LIN {X 0,Y 488.816,Z 673.843,A -85,B 0,C 180,E1 23597.214,E2 23597.214} C_VEL
LIN {X 0,Y 488.827,Z 673.82,A -85,B 0,C 180,E1 23593.605,E2 23593.605} C_VEL
LIN {X 0,Y 488.821,Z 673.843,A -85,B 0,C 180,E1 23590.012,E2 23590.012} C_VEL
LIN {X 0,Y 488.815,Z 673.84,A -85,B 0,C 180,E1 23586.459,E2 23586.459} C_VEL
LIN {X 0,Y 488.829,Z 673.833,A -85,B 0,C 180,E1 23582.931,E2 23582.931} C_VEL
LIN {X 0,Y 488.826,Z 673.843,A -85,B 0,C 180,E1 23579.297,E2 23579.297} C_VEL
LIN {X 0,Y 488.815,Z 673.842,A -85,B 0,C 180,E1 23575.659,E2 23575.659} C_VEL
LIN {X 0,Y 488.835,Z 673.84,A -85,B 0,C 180,E1 23572.123,E2 23572.123} C_VEL
LIN {X 0,Y 488.826,Z 673.833,A -85,B 0,C 180,E1 23568.556,E2 23568.556} C_VEL
LIN {X 0,Y 488.817,Z 673.838,A -85,B 0,C 180,E1 23564.943,E2 23564.943} C_VEL
LIN {X 0,Y 488.831,Z 673.84,A -85,B 0,C 180,E1 23561.392,E2 23561.392} C_VEL
LIN {X 0,Y 488.831,Z 673.844,A -85,B 0,C 180,E1 23557.765,E2 23557.765} C_VEL
LIN {X 0,Y 488.817,Z 673.841,A -85,B 0,C 180,E1 23554.155,E2 23554.155} C_VEL
LIN {X 0,Y 488.824,Z 673.804,A -85,B 0,C 180,E1 23550.6,E2 23550.6} C_VEL
LIN {X 0,Y 488.83,Z 673.841,A -85,B 0,C 180,E1 23546.992,E2 23546.992} C_VEL
LIN {X 0,Y 488.813,Z 673.808,A -85,B 0,C 180,E1 23543.47,E2 23543.47} C_VEL
LIN {X 0,Y 488.822,Z 673.844,A -85,B 0,C 180,E1 23539.885,E2 23539.885} C_VEL
LIN {X 0,Y 488.822,Z 673.817,A -85,B 0,C 180,E1 23536.221,E2 23536.221} C_VEL
LIN {X 0,Y 488.818,Z 673.811,A -85,B 0,C 180,E1 23532.75,E2 23532.75} C_VEL
LIN {X 0,Y 488.863,Z 674.082,A -85,B 0,C 180,E1 23530.778,E2 23530.778} C_VEL
LIN {X 0,Y 489.222,Z 675.525,A -85,B 0,C 180,E1 23530.578,E2 23530.578} C_VEL
LIN {X 0,Y 491.282,Z 678.683,A -85,B 0,C 180,E1 23530.298,E2 23530.298} C_VEL
LIN {X 0,Y 492.455,Z 680.416,A -85,B 0,C 180,E1 23530.144,E2 23530.144} C_VEL
LIN {X 0,Y 504.755,Z 699.098,A -85,B 0,C 180,E1 23528.583,E2 23528.583} C_VEL
LIN {X 0,Y 508.963,Z 706.354,A -85,B 0,C 180,E1 23528.059,E2 23528.059} C_VEL
LIN {X 0,Y 508.656,Z 723.177,A -85,B 0,C 180,E1 23527.787,E2 23527.787} C_VEL
LIN {X 0,Y 507.74,Z 730.874,A -85,B 0,C 180,E1 23527.733,E2 23527.733} C_VEL
LIN {X 0,Y 502.491,Z 751.441,A -85,B 0,C 180,E1 23527.848,E2 23527.848} C_VEL
LIN {X 0,Y 501.776,Z 758.046,A -85,B 0,C 180,E1 23527.795,E2 23527.795} C_VEL
LIN {X 0,Y 498.715,Z 918.69,A -85,B 0,C 180,E1 23525.17,E2 23525.17} C_VEL
LIN {X 0,Y 497.797,Z 939.753,A -85,B 0,C 180,E1 23524.625,E2 23524.625} C_VEL
LIN {X 0,Y 496.535,Z 960.944,A -85,B 0,C 180,E1 23523.867,E2 23523.867} C_VEL
LIN {X 0,Y 495.132,Z 980.222,A -85,B 0,C 180,E1 23522.97,E2 23522.97} C_VEL
LIN {X 0,Y 493.404,Z 999.351,A -85,B 0,C 180,E1 23521.862,E2 23521.862} C_VEL
LIN {X 0,Y 491.542,Z 1017.892,A -85,B 0,C 180,E1 23520.565,E2 23520.565} C_VEL
LIN {X 0,Y 489.26,Z 1039.477,A -85,B 0,C 180,E1 23518.752,E2 23518.752} C_VEL
LIN {X 0,Y 487.476,Z 1057.114,A -85,B 0,C 180,E1 23517.02,E2 23517.02} C_VEL
LIN {X 0,Y 485.787,Z 1073.337,A -85,B 0,C 180,E1 23515.151,E2 23515.151} C_VEL
LIN {X 0,Y 484.181,Z 1089.575,A -85,B 0,C 180,E1 23512.972,E2 23512.972} C_VEL
LIN {X 0,Y 482.951,Z 1103.101,A -85,B 0,C 180,E1 23510.86,E2 23510.86} C_VEL
LIN {X 0,Y 481.889,Z 1115.864,A -85,B 0,C 180,E1 23508.508,E2 23508.508} C_VEL
LIN {X 0,Y 481.077,Z 1127.142,A -85,B 0,C 180,E1 23506.046,E2 23506.046} C_VEL
LIN {X 0,Y 480.546,Z 1136.521,A -85,B 0,C 180,E1 23503.598,E2 23503.598} C_VEL
LIN {X 0,Y 480.213,Z 1144.105,A -85,B 0,C 180,E1 23501.165,E2 23501.165} C_VEL
LIN {X 0,Y 480.02,Z 1150.307,A -85,B 0,C 180,E1 23498.625,E2 23498.625} C_VEL
LIN {X 0,Y 479.931,Z 1154.921,A -85,B 0,C 180,E1 23496.099,E2 23496.099} C_VEL
LIN {X 0,Y 479.903,Z 1157.803,A -85,B 0,C 180,E1 23493.642,E2 23493.642} C_VEL
LIN {X 0,Y 479.906,Z 1159.318,A -85,B 0,C 180,E1 23490.955,E2 23490.955} C_VEL
LIN {X 0,Y 479.899,Z 1159.222,A -85,B 0,C 180,E1 23488.448,E2 23488.448} C_VEL
LIN {X 0,Y 479.909,Z 1157.49,A -85,B 0,C 180,E1 23485.938,E2 23485.938} C_VEL
LIN {X 0,Y 479.957,Z 1154.096,A -85,B 0,C 180,E1 23483.301,E2 23483.301} C_VEL
LIN {X 0,Y 480.049,Z 1149.377,A -85,B 0,C 180,E1 23480.845,E2 23480.845} C_VEL
LIN {X 0,Y 480.248,Z 1142.952,A -85,B 0,C 180,E1 23478.349,E2 23478.349} C_VEL
LIN {X 0,Y 480.611,Z 1135.144,A -85,B 0,C 180,E1 23475.913,E2 23475.913} C_VEL
LIN {X 0,Y 481.183,Z 1125.455,A -85,B 0,C 180,E1 23473.461,E2 23473.461} C_VEL
LIN {X 0,Y 482.017,Z 1114.139,A -85,B 0,C 180,E1 23471.066,E2 23471.066} C_VEL
LIN {X 0,Y 483.099,Z 1101.37,A -85,B 0,C 180,E1 23468.766,E2 23468.766} C_VEL
LIN {X 0,Y 484.384,Z 1087.622,A -85,B 0,C 180,E1 23466.652,E2 23466.652} C_VEL
LIN {X 0,Y 485.917,Z 1072.033,A -85,B 0,C 180,E1 23464.598,E2 23464.598} C_VEL
LIN {X 0,Y 487.685,Z 1054.909,A -85,B 0,C 180,E1 23462.662,E2 23462.662} C_VEL
LIN {X 0,Y 489.516,Z 1037.232,A -85,B 0,C 180,E1 23460.952,E2 23460.952} C_VEL
LIN {X 0,Y 491.779,Z 1015.791,A -85,B 0,C 180,E1 23459.18,E2 23459.18} C_VEL
LIN {X 0,Y 493.569,Z 997.713,A -85,B 0,C 180,E1 23457.945,E2 23457.945} C_VEL
LIN {X 0,Y 495.278,Z 978.123,A -85,B 0,C 180,E1 23456.834,E2 23456.834} C_VEL
LIN {X 0,Y 496.775,Z 957.74,A -85,B 0,C 180,E1 23455.908,E2 23455.908} C_VEL
LIN {X 0,Y 497.935,Z 937.311,A -85,B 0,C 180,E1 23455.213,E2 23455.213} C_VEL
LIN {X 0,Y 498.778,Z 915.593,A -85,B 0,C 180,E1 23454.681,E2 23454.681} C_VEL
LIN {X 0,Y 502.686,Z 709.142,A -85,B 0,C 180,E1 23451.313,E2 23451.313} C_VEL
LIN {X 0,Y 491.973,Z 692.433,A -85,B 0,C 180,E1 23449.946,E2 23449.946} C_VEL
LIN {X 0,Y 486.203,Z 683.956,A -85,B 0,C 180,E1 23449.181,E2 23449.181} C_VEL
LIN {X 0,Y 483.57,Z 679.859,A -85,B 0,C 180,E1 23448.819,E2 23448.819} C_VEL
LIN {X 0,Y 481.398,Z 676.823,A -85,B 0,C 180,E1 23448.52,E2 23448.52} C_VEL
LIN {X 0,Y 480.963,Z 675.357,A -85,B 0,C 180,E1 23448.364,E2 23448.364} C_VEL
LIN {X 0,Y 480.888,Z 674.825,A -85,B 0,C 180,E1 23448.104,E2 23448.104} C_VEL
LIN {X 0,Y 480.883,Z 674.824,A -85,B 0,C 180,E1 23444.483,E2 23444.483} C_VEL
LIN {X 0,Y 480.879,Z 674.818,A -85,B 0,C 180,E1 23440.917,E2 23440.917} C_VEL
LIN {X 0,Y 480.879,Z 674.795,A -85,B 0,C 180,E1 23437.383,E2 23437.383} C_VEL
LIN {X 0,Y 480.886,Z 674.832,A -85,B 0,C 180,E1 23433.721,E2 23433.721} C_VEL
LIN {X 0,Y 480.873,Z 674.785,A -85,B 0,C 180,E1 23430.073,E2 23430.073} C_VEL
LIN {X 0,Y 480.89,Z 674.835,A -85,B 0,C 180,E1 23426.42,E2 23426.42} C_VEL
LIN {X 0,Y 480.888,Z 674.83,A -85,B 0,C 180,E1 23422.751,E2 23422.751} C_VEL
LIN {X 0,Y 480.881,Z 674.827,A -85,B 0,C 180,E1 23419.179,E2 23419.179} C_VEL
LIN {X 0,Y 480.89,Z 674.823,A -85,B 0,C 180,E1 23415.558,E2 23415.558} C_VEL
LIN {X 0,Y 480.89,Z 674.823,A -85,B 0,C 180,E1 23411.879,E2 23411.879} C_VEL
LIN {X 0,Y 480.888,Z 674.831,A -85,B 0,C 180,E1 23408.245,E2 23408.245} C_VEL
LIN {X 0,Y 480.881,Z 674.831,A -85,B 0,C 180,E1 23404.532,E2 23404.532} C_VEL
LIN {X 0,Y 480.882,Z 674.827,A -85,B 0,C 180,E1 23400.953,E2 23400.953} C_VEL
LIN {X 0,Y 480.887,Z 674.821,A -85,B 0,C 180,E1 23397.378,E2 23397.378} C_VEL
LIN {X 0,Y 480.881,Z 674.828,A -85,B 0,C 180,E1 23393.793,E2 23393.793} C_VEL
LIN {X 0,Y 480.88,Z 674.834,A -85,B 0,C 180,E1 23390.184,E2 23390.184} C_VEL
LIN {X 0,Y 480.889,Z 674.805,A -85,B 0,C 180,E1 23386.534,E2 23386.534} C_VEL
LIN {X 0,Y 480.88,Z 674.831,A -85,B 0,C 180,E1 23382.952,E2 23382.952} C_VEL
LIN {X 0,Y 480.881,Z 674.827,A -85,B 0,C 180,E1 23379.301,E2 23379.301} C_VEL
LIN {X 0,Y 480.885,Z 674.812,A -85,B 0,C 180,E1 23375.69,E2 23375.69} C_VEL
LIN {X 0,Y 480.88,Z 674.834,A -85,B 0,C 180,E1 23372.085,E2 23372.085} C_VEL
LIN {X 0,Y 480.883,Z 674.834,A -85,B 0,C 180,E1 23368.479,E2 23368.479} C_VEL
LIN {X 0,Y 480.884,Z 674.828,A -85,B 0,C 180,E1 23364.796,E2 23364.796} C_VEL
LIN {X 0,Y 480.879,Z 674.826,A -85,B 0,C 180,E1 23361.232,E2 23361.232} C_VEL
LIN {X 0,Y 480.926,Z 675.033,A -85,B 0,C 180,E1 23358.576,E2 23358.576} C_VEL
LIN {X 0,Y 481.641,Z 677.323,A -85,B 0,C 180,E1 23358.212,E2 23358.212} C_VEL
LIN {X 0,Y 485.38,Z 684.871,A -85,B 0,C 180,E1 23357.165,E2 23357.165} C_VEL
LIN {X 0,Y 493.477,Z 702.425,A -85,B 0,C 180,E1 23354.917,E2 23354.917} C_VEL
LIN {X 0,Y 500.18,Z 718.461,A -85,B 0,C 180,E1 23353.052,E2 23353.052} C_VEL
LIN {X 0,Y 498.543,Z 751.608,A -85,B 0,C 180,E1 23350.747,E2 23350.747} C_VEL
LIN {X 0,Y 503.202,Z 783.353,A -85,B 0,C 180,E1 23349.737,E2 23349.737} C_VEL
LIN {X 0,Y 499.245,Z 1014.919,A -85,B 0,C 180,E1 23346.023,E2 23346.023} C_VEL
LIN {X 0,Y 498.268,Z 1064.193,A -85,B 0,C 180,E1 23345.211,E2 23345.211} C_VEL
LIN {X 0,Y 497.277,Z 1085.455,A -85,B 0,C 180,E1 23344.667,E2 23344.667} C_VEL
LIN {X 0,Y 495.928,Z 1108.008,A -85,B 0,C 180,E1 23343.879,E2 23343.879} C_VEL
LIN {X 0,Y 494.538,Z 1128.786,A -85,B 0,C 180,E1 23342.946,E2 23342.946} C_VEL
LIN {X 0,Y 492.887,Z 1149.43,A -85,B 0,C 180,E1 23341.792,E2 23341.792} C_VEL
LIN {X 0,Y 491.158,Z 1170.163,A -85,B 0,C 180,E1 23340.395,E2 23340.395} C_VEL
LIN {X 0,Y 489.454,Z 1187.758,A -85,B 0,C 180,E1 23338.955,E2 23338.955} C_VEL
LIN {X 0,Y 487.607,Z 1205.704,A -85,B 0,C 180,E1 23337.21,E2 23337.21} C_VEL
LIN {X 0,Y 485.852,Z 1222.673,A -85,B 0,C 180,E1 23335.278,E2 23335.278} C_VEL
LIN {X 0,Y 484.33,Z 1238.179,A -85,B 0,C 180,E1 23333.222,E2 23333.222} C_VEL
LIN {X 0,Y 482.996,Z 1252.633,A -85,B 0,C 180,E1 23330.985,E2 23330.985} C_VEL
LIN {X 0,Y 481.962,Z 1264.819,A -85,B 0,C 180,E1 23328.756,E2 23328.756} C_VEL
LIN {X 0,Y 481.114,Z 1276.544,A -85,B 0,C 180,E1 23326.234,E2 23326.234} C_VEL
LIN {X 0,Y 480.56,Z 1286.261,A -85,B 0,C 180,E1 23323.72,E2 23323.72} C_VEL
LIN {X 0,Y 480.216,Z 1293.884,A -85,B 0,C 180,E1 23321.286,E2 23321.286} C_VEL
LIN {X 0,Y 480.023,Z 1300.146,A -85,B 0,C 180,E1 23318.746,E2 23318.746} C_VEL
LIN {X 0,Y 479.935,Z 1304.636,A -85,B 0,C 180,E1 23316.339,E2 23316.339} C_VEL
LIN {X 0,Y 479.902,Z 1307.673,A -85,B 0,C 180,E1 23313.823,E2 23313.823} C_VEL
LIN {X 0,Y 479.907,Z 1309.281,A -85,B 0,C 180,E1 23311.194,E2 23311.194} C_VEL
LIN {X 0,Y 479.907,Z 1309.281,A -85,B 0,C 180,E1 23308.806,E2 23308.806} C_VEL
LIN {X 0,Y 479.902,Z 1307.671,A -85,B 0,C 180,E1 23306.177,E2 23306.177} C_VEL
LIN {X 0,Y 479.935,Z 1304.633,A -85,B 0,C 180,E1 23303.661,E2 23303.661} C_VEL
LIN {X 0,Y 480.023,Z 1300.145,A -85,B 0,C 180,E1 23301.254,E2 23301.254} C_VEL
LIN {X 0,Y 480.23,Z 1293.528,A -85,B 0,C 180,E1 23298.592,E2 23298.592} C_VEL
LIN {X 0,Y 480.582,Z 1285.851,A -85,B 0,C 180,E1 23296.158,E2 23296.158} C_VEL
LIN {X 0,Y 481.132,Z 1276.296,A -85,B 0,C 180,E1 23293.708,E2 23293.708} C_VEL
LIN {X 0,Y 481.961,Z 1264.819,A -85,B 0,C 180,E1 23291.243,E2 23291.243} C_VEL
LIN {X 0,Y 483.001,Z 1252.568,A -85,B 0,C 180,E1 23289.004,E2 23289.004} C_VEL
LIN {X 0,Y 484.33,Z 1238.179,A -85,B 0,C 180,E1 23286.778,E2 23286.778} C_VEL
LIN {X 0,Y 485.853,Z 1222.674,A -85,B 0,C 180,E1 23284.722,E2 23284.722} C_VEL
LIN {X 0,Y 487.606,Z 1205.703,A -85,B 0,C 180,E1 23282.79,E2 23282.79} C_VEL
LIN {X 0,Y 489.455,Z 1187.76,A -85,B 0,C 180,E1 23281.045,E2 23281.045} C_VEL
LIN {X 0,Y 491.16,Z 1170.167,A -85,B 0,C 180,E1 23279.605,E2 23279.605} C_VEL
LIN {X 0,Y 492.887,Z 1149.435,A -85,B 0,C 180,E1 23278.208,E2 23278.208} C_VEL
LIN {X 0,Y 494.567,Z 1128.4,A -85,B 0,C 180,E1 23277.034,E2 23277.034} C_VEL
LIN {X 0,Y 495.983,Z 1107.264,A -85,B 0,C 180,E1 23276.09,E2 23276.09} C_VEL
LIN {X 0,Y 497.313,Z 1084.768,A -85,B 0,C 180,E1 23275.312,E2 23275.312} C_VEL
LIN {X 0,Y 498.303,Z 1063.308,A -85,B 0,C 180,E1 23274.77,E2 23274.77} C_VEL
LIN {X 0,Y 499.952,Z 971.981,A -85,B 0,C 180,E1 23273.295,E2 23273.295} C_VEL
LIN {X 0,Y 503.149,Z 781.671,A -85,B 0,C 180,E1 23270.228,E2 23270.228} C_VEL
LIN {X 0,Y 498.478,Z 750.795,A -85,B 0,C 180,E1 23269.217,E2 23269.217} C_VEL
LIN {X 0,Y 500.171,Z 717.88,A -85,B 0,C 180,E1 23266.903,E2 23266.903} C_VEL
LIN {X 0,Y 489.861,Z 694.265,A -85,B 0,C 180,E1 23264.074,E2 23264.074} C_VEL
LIN {X 0,Y 482.531,Z 678.757,A -85,B 0,C 180,E1 23262.012,E2 23262.012} C_VEL
LIN {X 0,Y 480.927,Z 675.052,A -85,B 0,C 180,E1 23261.461,E2 23261.461} C_VEL
LIN {X 0,Y 480.876,Z 674.825,A -85,B 0,C 180,E1 23258.744,E2 23258.744} C_VEL
LIN {X 0,Y 480.885,Z 674.827,A -85,B 0,C 180,E1 23255.165,E2 23255.165} C_VEL
LIN {X 0,Y 480.88,Z 674.834,A -85,B 0,C 180,E1 23251.459,E2 23251.459} C_VEL
LIN {X 0,Y 480.881,Z 674.834,A -85,B 0,C 180,E1 23247.893,E2 23247.893} C_VEL
LIN {X 0,Y 480.886,Z 674.813,A -85,B 0,C 180,E1 23244.18,E2 23244.18} C_VEL
LIN {X 0,Y 480.879,Z 674.824,A -85,B 0,C 180,E1 23240.572,E2 23240.572} C_VEL
LIN {X 0,Y 480.884,Z 674.83,A -85,B 0,C 180,E1 23236.923,E2 23236.923} C_VEL
LIN {X 0,Y 480.881,Z 674.805,A -85,B 0,C 180,E1 23233.221,E2 23233.221} C_VEL
LIN {X 0,Y 480.879,Z 674.836,A -85,B 0,C 180,E1 23229.696,E2 23229.696} C_VEL
LIN {X 0,Y 480.885,Z 674.828,A -85,B 0,C 180,E1 23226.087,E2 23226.087} C_VEL
LIN {X 0,Y 480.881,Z 674.823,A -85,B 0,C 180,E1 23222.383,E2 23222.383} C_VEL
LIN {X 0,Y 480.889,Z 674.823,A -85,B 0,C 180,E1 23218.808,E2 23218.808} C_VEL
LIN {X 0,Y 480.887,Z 674.833,A -85,B 0,C 180,E1 23215.11,E2 23215.11} C_VEL
LIN {X 0,Y 480.879,Z 674.831,A -85,B 0,C 180,E1 23211.51,E2 23211.51} C_VEL
LIN {X 0,Y 480.894,Z 674.825,A -85,B 0,C 180,E1 23207.878,E2 23207.878} C_VEL
LIN {X 0,Y 480.89,Z 674.822,A -85,B 0,C 180,E1 23204.287,E2 23204.287} C_VEL
LIN {X 0,Y 480.879,Z 674.828,A -85,B 0,C 180,E1 23200.695,E2 23200.695} C_VEL
LIN {X 0,Y 480.891,Z 674.828,A -85,B 0,C 180,E1 23197.08,E2 23197.08} C_VEL
LIN {X 0,Y 480.892,Z 674.835,A -85,B 0,C 180,E1 23193.382,E2 23193.382} C_VEL
LIN {X 0,Y 480.869,Z 674.786,A -85,B 0,C 180,E1 23189.789,E2 23189.789} C_VEL
LIN {X 0,Y 480.891,Z 674.831,A -85,B 0,C 180,E1 23186.136,E2 23186.136} C_VEL
LIN {X 0,Y 480.878,Z 674.796,A -85,B 0,C 180,E1 23182.467,E2 23182.467} C_VEL
LIN {X 0,Y 480.877,Z 674.817,A -85,B 0,C 180,E1 23178.925,E2 23178.925} C_VEL
LIN {X 0,Y 480.889,Z 674.828,A -85,B 0,C 180,E1 23175.321,E2 23175.321} C_VEL
LIN {X 0,Y 480.892,Z 674.933,A -85,B 0,C 180,E1 23171.651,E2 23171.651} C_VEL
LIN {X 0,Y 481.211,Z 676.309,A -85,B 0,C 180,E1 23171.425,E2 23171.425} C_VEL
LIN {X 0,Y 483.113,Z 679.426,A -85,B 0,C 180,E1 23171.148,E2 23171.148} C_VEL
LIN {X 0,Y 484.393,Z 681.057,A -85,B 0,C 180,E1 23170.978,E2 23170.978} C_VEL
LIN {X 0,Y 499.081,Z 703.249,A -85,B 0,C 180,E1 23169.052,E2 23169.052} C_VEL
LIN {X 0,Y 502.72,Z 709.568,A -85,B 0,C 180,E1 23168.586,E2 23168.586} C_VEL
LIN {X 0,Y 501.776,Z 758.046,A -85,B 0,C 180,E1 23167.795,E2 23167.795} C_VEL
LIN {X 0,Y 500.849,Z 765.743,A -85,B 0,C 180,E1 23167.742,E2 23167.742} C_VEL
LIN {X 0,Y 495.581,Z 786.303,A -85,B 0,C 180,E1 23167.86,E2 23167.86} C_VEL
LIN {X 0,Y 494.861,Z 792.908,A -85,B 0,C 180,E1 23167.807,E2 23167.807} C_VEL
LIN {X 0,Y 492.27,Z 920.125,A -85,B 0,C 180,E1 23165.7,E2 23165.7} C_VEL
LIN {X 0,Y 491.313,Z 941.343,A -85,B 0,C 180,E1 23165.143,E2 23165.143} C_VEL
LIN {X 0,Y 489.963,Z 963.073,A -85,B 0,C 180,E1 23164.349,E2 23164.349} C_VEL
LIN {X 0,Y 488.452,Z 982.868,A -85,B 0,C 180,E1 23163.41,E2 23163.41} C_VEL
LIN {X 0,Y 486.63,Z 1001.725,A -85,B 0,C 180,E1 23162.289,E2 23162.289} C_VEL
LIN {X 0,Y 484.584,Z 1020.851,A -85,B 0,C 180,E1 23160.914,E2 23160.914} C_VEL
LIN {X 0,Y 482.545,Z 1038.387,A -85,B 0,C 180,E1 23159.41,E2 23159.41} C_VEL
LIN {X 0,Y 480.437,Z 1054.914,A -85,B 0,C 180,E1 23157.718,E2 23157.718} C_VEL
LIN {X 0,Y 478.341,Z 1073.262,A -85,B 0,C 180,E1 23155.581,E2 23155.581} C_VEL
LIN {X 0,Y 476.695,Z 1088.735,A -85,B 0,C 180,E1 23153.485,E2 23153.485} C_VEL
LIN {X 0,Y 475.281,Z 1102.849,A -85,B 0,C 180,E1 23151.259,E2 23151.259} C_VEL
LIN {X 0,Y 474.142,Z 1115.231,A -85,B 0,C 180,E1 23148.95,E2 23148.95} C_VEL
LIN {X 0,Y 473.225,Z 1126.757,A -85,B 0,C 180,E1 23146.415,E2 23146.415} C_VEL
LIN {X 0,Y 472.634,Z 1136.117,A -85,B 0,C 180,E1 23143.955,E2 23143.955} C_VEL
LIN {X 0,Y 472.258,Z 1143.754,A -85,B 0,C 180,E1 23141.479,E2 23141.479} C_VEL
LIN {X 0,Y 472.045,Z 1150.054,A -85,B 0,C 180,E1 23138.895,E2 23138.895} C_VEL
LIN {X 0,Y 471.94,Z 1154.758,A -85,B 0,C 180,E1 23136.325,E2 23136.325} C_VEL
LIN {X 0,Y 471.902,Z 1157.746,A -85,B 0,C 180,E1 23133.766,E2 23133.766} C_VEL
LIN {X 0,Y 471.908,Z 1159.295,A -85,B 0,C 180,E1 23131.093,E2 23131.093} C_VEL
LIN {X 0,Y 471.907,Z 1159.267,A -85,B 0,C 180,E1 23128.665,E2 23128.665} C_VEL
LIN {X 0,Y 471.906,Z 1157.716,A -85,B 0,C 180,E1 23126.112,E2 23126.112} C_VEL
LIN {X 0,Y 471.949,Z 1154.657,A -85,B 0,C 180,E1 23123.521,E2 23123.521} C_VEL
LIN {X 0,Y 472.048,Z 1149.984,A -85,B 0,C 180,E1 23120.982,E2 23120.982} C_VEL
LIN {X 0,Y 472.271,Z 1143.303,A -85,B 0,C 180,E1 23118.274,E2 23118.274} C_VEL
LIN {X 0,Y 472.663,Z 1135.588,A -85,B 0,C 180,E1 23115.796,E2 23115.796} C_VEL
LIN {X 0,Y 473.277,Z 1125.966,A -85,B 0,C 180,E1 23113.303,E2 23113.303} C_VEL
LIN {X 0,Y 474.206,Z 1114.407,A -85,B 0,C 180,E1 23110.797,E2 23110.797} C_VEL
LIN {X 0,Y 475.346,Z 1102.136,A -85,B 0,C 180,E1 23108.532,E2 23108.532} C_VEL
LIN {X 0,Y 476.719,Z 1088.463,A -85,B 0,C 180,E1 23106.385,E2 23106.385} C_VEL
LIN {X 0,Y 478.4,Z 1072.735,A -85,B 0,C 180,E1 23104.263,E2 23104.263} C_VEL
LIN {X 0,Y 480.556,Z 1053.957,A -85,B 0,C 180,E1 23102.087,E2 23102.087} C_VEL
LIN {X 0,Y 482.686,Z 1037.225,A -85,B 0,C 180,E1 23100.395,E2 23100.395} C_VEL
LIN {X 0,Y 484.645,Z 1020.305,A -85,B 0,C 180,E1 23098.952,E2 23098.952} C_VEL
LIN {X 0,Y 486.703,Z 1001.044,A -85,B 0,C 180,E1 23097.577,E2 23097.577} C_VEL
LIN {X 0,Y 488.516,Z 981.99,A -85,B 0,C 180,E1 23096.455,E2 23096.455} C_VEL
LIN {X 0,Y 490.034,Z 962.107,A -85,B 0,C 180,E1 23095.52,E2 23095.52} C_VEL
LIN {X 0,Y 491.341,Z 940.901,A -85,B 0,C 180,E1 23094.754,E2 23094.754} C_VEL
LIN {X 0,Y 492.279,Z 919.721,A -85,B 0,C 180,E1 23094.202,E2 23094.202} C_VEL
LIN {X 0,Y 496.488,Z 712.422,A -85,B 0,C 180,E1 23090.774,E2 23090.774} C_VEL
LIN {X 0,Y 484.896,Z 694.452,A -85,B 0,C 180,E1 23089.247,E2 23089.247} C_VEL
LIN {X 0,Y 478.519,Z 685.19,A -85,B 0,C 180,E1 23088.371,E2 23088.371} C_VEL
LIN {X 0,Y 475.607,Z 680.806,A -85,B 0,C 180,E1 23087.956,E2 23087.956} C_VEL
LIN {X 0,Y 473.496,Z 677.855,A -85,B 0,C 180,E1 23087.653,E2 23087.653} C_VEL
LIN {X 0,Y 472.994,Z 676.129,A -85,B 0,C 180,E1 23087.435,E2 23087.435} C_VEL
LIN {X 0,Y 472.937,Z 675.792,A -85,B 0,C 180,E1 23086.482,E2 23086.482} C_VEL
LIN {X 0,Y 472.94,Z 675.78,A -85,B 0,C 180,E1 23082.903,E2 23082.903} C_VEL
LIN {X 0,Y 472.952,Z 675.817,A -85,B 0,C 180,E1 23079.206,E2 23079.206} C_VEL
LIN {X 0,Y 472.937,Z 675.795,A -85,B 0,C 180,E1 23075.519,E2 23075.519} C_VEL
LIN {X 0,Y 472.946,Z 675.799,A -85,B 0,C 180,E1 23071.906,E2 23071.906} C_VEL
LIN {X 0,Y 472.941,Z 675.797,A -85,B 0,C 180,E1 23068.266,E2 23068.266} C_VEL
LIN {X 0,Y 472.952,Z 675.811,A -85,B 0,C 180,E1 23064.612,E2 23064.612} C_VEL
LIN {X 0,Y 472.956,Z 675.813,A -85,B 0,C 180,E1 23060.933,E2 23060.933} C_VEL
LIN {X 0,Y 472.939,Z 675.817,A -85,B 0,C 180,E1 23057.343,E2 23057.343} C_VEL
LIN {X 0,Y 472.952,Z 675.824,A -85,B 0,C 180,E1 23053.697,E2 23053.697} C_VEL
LIN {X 0,Y 472.954,Z 675.815,A -85,B 0,C 180,E1 23049.983,E2 23049.983} C_VEL
LIN {X 0,Y 472.938,Z 675.807,A -85,B 0,C 180,E1 23046.434,E2 23046.434} C_VEL
LIN {X 0,Y 472.947,Z 675.809,A -85,B 0,C 180,E1 23042.787,E2 23042.787} C_VEL
LIN {X 0,Y 472.955,Z 675.824,A -85,B 0,C 180,E1 23039.152,E2 23039.152} C_VEL
LIN {X 0,Y 472.94,Z 675.819,A -85,B 0,C 180,E1 23035.514,E2 23035.514} C_VEL
LIN {X 0,Y 472.95,Z 675.813,A -85,B 0,C 180,E1 23031.857,E2 23031.857} C_VEL
LIN {X 0,Y 472.938,Z 675.802,A -85,B 0,C 180,E1 23028.167,E2 23028.167} C_VEL
LIN {X 0,Y 472.947,Z 675.818,A -85,B 0,C 180,E1 23024.551,E2 23024.551} C_VEL
LIN {X 0,Y 472.94,Z 675.793,A -85,B 0,C 180,E1 23020.872,E2 23020.872} C_VEL
LIN {X 0,Y 472.938,Z 675.818,A -85,B 0,C 180,E1 23017.239,E2 23017.239} C_VEL
LIN {X 0,Y 472.947,Z 675.819,A -85,B 0,C 180,E1 23013.508,E2 23013.508} C_VEL
LIN {X 0,Y 472.938,Z 675.801,A -85,B 0,C 180,E1 23009.844,E2 23009.844} C_VEL
LIN {X 0,Y 472.947,Z 675.8,A -85,B 0,C 180,E1 23006.183,E2 23006.183} C_VEL
LIN {X 0,Y 472.94,Z 675.804,A -85,B 0,C 180,E1 23002.492,E2 23002.492} C_VEL
LIN {X 0,Y 472.985,Z 676.069,A -85,B 0,C 180,E1 22999.381,E2 22999.381} C_VEL
LIN {X 0,Y 474.306,Z 679.352,A -85,B 0,C 180,E1 22998.875,E2 22998.875} C_VEL
LIN {X 0,Y 481.226,Z 693.654,A -85,B 0,C 180,E1 22996.877,E2 22996.877} C_VEL
LIN {X 0,Y 489.916,Z 713.159,A -85,B 0,C 180,E1 22994.414,E2 22994.414} C_VEL
LIN {X 0,Y 493.417,Z 721.382,A -85,B 0,C 180,E1 22993.442,E2 22993.442} C_VEL
LIN {X 0,Y 491.892,Z 750.061,A -85,B 0,C 180,E1 22991.418,E2 22991.418} C_VEL
LIN {X 0,Y 496.921,Z 784.692,A -85,B 0,C 180,E1 22990.291,E2 22990.291} C_VEL
LIN {X 0,Y 492.662,Z 1016.075,A -85,B 0,C 180,E1 22986.537,E2 22986.537} C_VEL
LIN {X 0,Y 491.642,Z 1062.974,A -85,B 0,C 180,E1 22985.752,E2 22985.752} C_VEL
LIN {X 0,Y 490.544,Z 1084.634,A -85,B 0,C 180,E1 22985.192,E2 22985.192} C_VEL
LIN {X 0,Y 489.122,Z 1106.554,A -85,B 0,C 180,E1 22984.416,E2 22984.416} C_VEL
LIN {X 0,Y 487.522,Z 1127.997,A -85,B 0,C 180,E1 22983.441,E2 22983.441} C_VEL
LIN {X 0,Y 485.777,Z 1148.406,A -85,B 0,C 180,E1 22982.283,E2 22982.283} C_VEL
LIN {X 0,Y 483.916,Z 1168.797,A -85,B 0,C 180,E1 22980.893,E2 22980.893} C_VEL
LIN {X 0,Y 482.047,Z 1188.505,A -85,B 0,C 180,E1 22979.307,E2 22979.307} C_VEL
LIN {X 0,Y 480.548,Z 1203.264,A -85,B 0,C 180,E1 22977.913,E2 22977.913} C_VEL
LIN {X 0,Y 478.701,Z 1220.139,A -85,B 0,C 180,E1 22976.015,E2 22976.015} C_VEL
LIN {X 0,Y 477.006,Z 1235.883,A -85,B 0,C 180,E1 22973.95,E2 22973.95} C_VEL
LIN {X 0,Y 475.507,Z 1250.323,A -85,B 0,C 180,E1 22971.72,E2 22971.72} C_VEL
LIN {X 0,Y 474.274,Z 1263.548,A -85,B 0,C 180,E1 22969.328,E2 22969.328} C_VEL
LIN {X 0,Y 473.355,Z 1274.977,A -85,B 0,C 180,E1 22966.891,E2 22966.891} C_VEL
LIN {X 0,Y 472.702,Z 1284.853,A -85,B 0,C 180,E1 22964.36,E2 22964.36} C_VEL
LIN {X 0,Y 472.293,Z 1292.823,A -85,B 0,C 180,E1 22961.85,E2 22961.85} C_VEL
LIN {X 0,Y 472.063,Z 1299.421,A -85,B 0,C 180,E1 22959.245,E2 22959.245} C_VEL
LIN {X 0,Y 471.96,Z 1304.019,A -85,B 0,C 180,E1 22956.813,E2 22956.813} C_VEL
LIN {X 0,Y 471.907,Z 1307.446,A -85,B 0,C 180,E1 22954.131,E2 22954.131} C_VEL
LIN {X 0,Y 471.896,Z 1309.209,A -85,B 0,C 180,E1 22951.578,E2 22951.578} C_VEL
LIN {X 0,Y 471.906,Z 1309.326,A -85,B 0,C 180,E1 22949.029,E2 22949.029} C_VEL
LIN {X 0,Y 471.903,Z 1307.865,A -85,B 0,C 180,E1 22946.321,E2 22946.321} C_VEL
LIN {X 0,Y 471.931,Z 1304.979,A -85,B 0,C 180,E1 22943.797,E2 22943.797} C_VEL
LIN {X 0,Y 472.029,Z 1300.399,A -85,B 0,C 180,E1 22941.228,E2 22941.228} C_VEL
LIN {X 0,Y 472.238,Z 1294.235,A -85,B 0,C 180,E1 22938.644,E2 22938.644} C_VEL
LIN {X 0,Y 472.605,Z 1286.666,A -85,B 0,C 180,E1 22936.169,E2 22936.169} C_VEL
LIN {X 0,Y 473.212,Z 1276.955,A -85,B 0,C 180,E1 22933.589,E2 22933.589} C_VEL
LIN {X 0,Y 474.069,Z 1266.088,A -85,B 0,C 180,E1 22931.175,E2 22931.175} C_VEL
LIN {X 0,Y 475.155,Z 1254.059,A -85,B 0,C 180,E1 22928.911,E2 22928.911} C_VEL
LIN {X 0,Y 476.477,Z 1240.713,A -85,B 0,C 180,E1 22926.766,E2 22926.766} C_VEL
LIN {X 0,Y 478.089,Z 1225.714,A -85,B 0,C 180,E1 22924.68,E2 22924.68} C_VEL
LIN {X 0,Y 479.92,Z 1209.246,A -85,B 0,C 180,E1 22922.721,E2 22922.721} C_VEL
LIN {X 0,Y 481.488,Z 1194.127,A -85,B 0,C 180,E1 22921.2,E2 22921.2} C_VEL
LIN {X 0,Y 483.389,Z 1174.738,A -85,B 0,C 180,E1 22919.552,E2 22919.552} C_VEL
LIN {X 0,Y 485.231,Z 1154.409,A -85,B 0,C 180,E1 22918.098,E2 22918.098} C_VEL
LIN {X 0,Y 487.007,Z 1134.2,A -85,B 0,C 180,E1 22916.893,E2 22916.893} C_VEL
LIN {X 0,Y 488.655,Z 1113.398,A -85,B 0,C 180,E1 22915.866,E2 22915.866} C_VEL
LIN {X 0,Y 490.145,Z 1091.17,A -85,B 0,C 180,E1 22915.013,E2 22915.013} C_VEL
LIN {X 0,Y 491.354,Z 1069.19,A -85,B 0,C 180,E1 22914.393,E2 22914.393} C_VEL
LIN {X 0,Y 492.151,Z 1045.544,A -85,B 0,C 180,E1 22913.936,E2 22913.936} C_VEL
LIN {X 0,Y 496.185,Z 822.336,A -85,B 0,C 180,E1 22910.324,E2 22910.324} C_VEL
LIN {X 0,Y 496.78,Z 782.531,A -85,B 0,C 180,E1 22909.656,E2 22909.656} C_VEL
LIN {X 0,Y 491.829,Z 749.318,A -85,B 0,C 180,E1 22908.55,E2 22908.55} C_VEL
LIN {X 0,Y 493.282,Z 721.075,A -85,B 0,C 180,E1 22906.522,E2 22906.522} C_VEL
LIN {X 0,Y 483.709,Z 698.95,A -85,B 0,C 180,E1 22903.825,E2 22903.825} C_VEL
LIN {X 0,Y 476.318,Z 683.416,A -85,B 0,C 180,E1 22901.715,E2 22901.715} C_VEL
LIN {X 0,Y 474.297,Z 679.327,A -85,B 0,C 180,E1 22901.126,E2 22901.126} C_VEL
LIN {X 0,Y 472.974,Z 676.014,A -85,B 0,C 180,E1 22900.606,E2 22900.606} C_VEL
LIN {X 0,Y 472.948,Z 675.806,A -85,B 0,C 180,E1 22897.05,E2 22897.05} C_VEL
LIN {X 0,Y 472.938,Z 675.803,A -85,B 0,C 180,E1 22893.378,E2 22893.378} C_VEL
LIN {X 0,Y 472.945,Z 675.797,A -85,B 0,C 180,E1 22889.789,E2 22889.789} C_VEL
LIN {X 0,Y 472.94,Z 675.813,A -85,B 0,C 180,E1 22886.087,E2 22886.087} C_VEL
LIN {X 0,Y 472.939,Z 675.82,A -85,B 0,C 180,E1 22882.498,E2 22882.498} C_VEL
LIN {X 0,Y 472.945,Z 675.793,A -85,B 0,C 180,E1 22878.872,E2 22878.872} C_VEL
LIN {X 0,Y 472.94,Z 675.816,A -85,B 0,C 180,E1 22875.198,E2 22875.198} C_VEL
LIN {X 0,Y 472.943,Z 675.805,A -85,B 0,C 180,E1 22871.586,E2 22871.586} C_VEL
LIN {X 0,Y 472.945,Z 675.812,A -85,B 0,C 180,E1 22867.898,E2 22867.898} C_VEL
LIN {X 0,Y 472.938,Z 675.818,A -85,B 0,C 180,E1 22864.243,E2 22864.243} C_VEL
LIN {X 0,Y 472.958,Z 675.823,A -85,B 0,C 180,E1 22860.605,E2 22860.605} C_VEL
LIN {X 0,Y 472.945,Z 675.812,A -85,B 0,C 180,E1 22856.97,E2 22856.97} C_VEL
LIN {X 0,Y 472.942,Z 675.806,A -85,B 0,C 180,E1 22853.323,E2 22853.323} C_VEL
LIN {X 0,Y 472.949,Z 675.813,A -85,B 0,C 180,E1 22849.648,E2 22849.648} C_VEL
LIN {X 0,Y 472.954,Z 675.823,A -85,B 0,C 180,E1 22846.008,E2 22846.008} C_VEL
LIN {X 0,Y 472.949,Z 675.819,A -85,B 0,C 180,E1 22842.276,E2 22842.276} C_VEL
LIN {X 0,Y 472.943,Z 675.816,A -85,B 0,C 180,E1 22838.677,E2 22838.677} C_VEL
LIN {X 0,Y 472.95,Z 675.812,A -85,B 0,C 180,E1 22835.083,E2 22835.083} C_VEL
LIN {X 0,Y 472.952,Z 675.79,A -85,B 0,C 180,E1 22831.459,E2 22831.459} C_VEL
LIN {X 0,Y 472.939,Z 675.807,A -85,B 0,C 180,E1 22827.807,E2 22827.807} C_VEL
LIN {X 0,Y 472.941,Z 675.792,A -85,B 0,C 180,E1 22824.272,E2 22824.272} C_VEL
LIN {X 0,Y 472.955,Z 675.818,A -85,B 0,C 180,E1 22820.638,E2 22820.638} C_VEL
LIN {X 0,Y 472.935,Z 675.782,A -85,B 0,C 180,E1 22816.931,E2 22816.931} C_VEL
LIN {X 0,Y 472.942,Z 675.79,A -85,B 0,C 180,E1 22813.343,E2 22813.343} C_VEL
LIN {X 0,Y 472.982,Z 676.068,A -85,B 0,C 180,E1 22812.487,E2 22812.487} C_VEL
LIN {X 0,Y 473.487,Z 677.842,A -85,B 0,C 180,E1 22812.256,E2 22812.256} C_VEL
LIN {X 0,Y 475.608,Z 680.81,A -85,B 0,C 180,E1 22811.952,E2 22811.952} C_VEL
LIN {X 0,Y 477.215,Z 683.359,A -85,B 0,C 180,E1 22811.719,E2 22811.719} C_VEL
LIN {X 0,Y 480.421,Z 687.944,A -85,B 0,C 180,E1 22811.273,E2 22811.273} C_VEL
LIN {X 0,Y 491.752,Z 704.844,A -85,B 0,C 180,E1 22809.751,E2 22809.751} C_VEL
LIN {X 0,Y 496.521,Z 712.769,A -85,B 0,C 180,E1 22809.126,E2 22809.126} C_VEL
LIN {X 0,Y 494.861,Z 792.908,A -85,B 0,C 180,E1 22807.807,E2 22807.807} C_VEL
LIN {X 0,Y 493.921,Z 800.607,A -85,B 0,C 180,E1 22807.754,E2 22807.754} C_VEL
LIN {X 0,Y 488.615,Z 821.161,A -85,B 0,C 180,E1 22807.878,E2 22807.878} C_VEL
LIN {X 0,Y 487.913,Z 827.764,A -85,B 0,C 180,E1 22807.822,E2 22807.822} C_VEL
LIN {X 0,Y 485.866,Z 921.688,A -85,B 0,C 180,E1 22806.242,E2 22806.242} C_VEL
LIN {X 0,Y 484.865,Z 942.972,A -85,B 0,C 180,E1 22805.673,E2 22805.673} C_VEL
LIN {X 0,Y 483.48,Z 964.482,A -85,B 0,C 180,E1 22804.876,E2 22804.876} C_VEL
LIN {X 0,Y 481.855,Z 984.74,A -85,B 0,C 180,E1 22803.9,E2 22803.9} C_VEL
LIN {X 0,Y 479.887,Z 1004.096,A -85,B 0,C 180,E1 22802.729,E2 22802.729} C_VEL
LIN {X 0,Y 477.748,Z 1022.953,A -85,B 0,C 180,E1 22801.343,E2 22801.343} C_VEL
LIN {X 0,Y 475.587,Z 1040.439,A -85,B 0,C 180,E1 22799.815,E2 22799.815} C_VEL
LIN {X 0,Y 473.368,Z 1056.895,A -85,B 0,C 180,E1 22798.1,E2 22798.1} C_VEL
LIN {X 0,Y 471.176,Z 1072.789,A -85,B 0,C 180,E1 22796.152,E2 22796.152} C_VEL
LIN {X 0,Y 468.653,Z 1092.962,A -85,B 0,C 180,E1 22793.246,E2 22793.246} C_VEL
LIN {X 0,Y 467.19,Z 1106.62,A -85,B 0,C 180,E1 22790.94,E2 22790.94} C_VEL
LIN {X 0,Y 466.022,Z 1118.953,A -85,B 0,C 180,E1 22788.5,E2 22788.5} C_VEL
LIN {X 0,Y 465.181,Z 1129.205,A -85,B 0,C 180,E1 22786.097,E2 22786.097} C_VEL
LIN {X 0,Y 464.585,Z 1138.146,A -85,B 0,C 180,E1 22783.567,E2 22783.567} C_VEL
LIN {X 0,Y 464.209,Z 1145.748,A -85,B 0,C 180,E1 22780.926,E2 22780.926} C_VEL
LIN {X 0,Y 464.017,Z 1151.328,A -85,B 0,C 180,E1 22778.425,E2 22778.425} C_VEL
LIN {X 0,Y 463.932,Z 1155.563,A -85,B 0,C 180,E1 22775.813,E2 22775.813} C_VEL
LIN {X 0,Y 463.909,Z 1158.306,A -85,B 0,C 180,E1 22773.212,E2 22773.212} C_VEL
LIN {X 0,Y 463.896,Z 1159.385,A -85,B 0,C 180,E1 22770.617,E2 22770.617} C_VEL
LIN {X 0,Y 463.907,Z 1158.976,A -85,B 0,C 180,E1 22767.9,E2 22767.9} C_VEL
LIN {X 0,Y 463.917,Z 1157.147,A -85,B 0,C 180,E1 22765.426,E2 22765.426} C_VEL
LIN {X 0,Y 463.958,Z 1153.68,A -85,B 0,C 180,E1 22762.82,E2 22762.82} C_VEL
LIN {X 0,Y 464.087,Z 1148.965,A -85,B 0,C 180,E1 22760.326,E2 22760.326} C_VEL
LIN {X 0,Y 464.343,Z 1142.594,A -85,B 0,C 180,E1 22757.818,E2 22757.818} C_VEL
LIN {X 0,Y 464.829,Z 1134.218,A -85,B 0,C 180,E1 22755.169,E2 22755.169} C_VEL
LIN {X 0,Y 465.561,Z 1124.412,A -85,B 0,C 180,E1 22752.632,E2 22752.632} C_VEL
LIN {X 0,Y 466.564,Z 1113.011,A -85,B 0,C 180,E1 22750.185,E2 22750.185} C_VEL
LIN {X 0,Y 467.953,Z 1099.325,A -85,B 0,C 180,E1 22747.695,E2 22747.695} C_VEL
LIN {X 0,Y 469.56,Z 1084.969,A -85,B 0,C 180,E1 22745.467,E2 22745.467} C_VEL
LIN {X 0,Y 471.855,Z 1068.081,A -85,B 0,C 180,E1 22743.138,E2 22743.138} C_VEL
LIN {X 0,Y 474.055,Z 1051.876,A -85,B 0,C 180,E1 22741.257,E2 22741.257} C_VEL
LIN {X 0,Y 476.249,Z 1035.097,A -85,B 0,C 180,E1 22739.606,E2 22739.606} C_VEL
LIN {X 0,Y 478.483,Z 1016.837,A -85,B 0,C 180,E1 22738.085,E2 22738.085} C_VEL
LIN {X 0,Y 480.496,Z 998.53,A -85,B 0,C 180,E1 22736.821,E2 22736.821} C_VEL
LIN {X 0,Y 482.26,Z 979.621,A -85,B 0,C 180,E1 22735.745,E2 22735.745} C_VEL
LIN {X 0,Y 483.882,Z 959.146,A -85,B 0,C 180,E1 22734.81,E2 22734.81} C_VEL
LIN {X 0,Y 485.112,Z 938.858,A -85,B 0,C 180,E1 22734.112,E2 22734.112} C_VEL
LIN {X 0,Y 485.981,Z 916.775,A -85,B 0,C 180,E1 22733.571,E2 22733.571} C_VEL
LIN {X 0,Y 490.327,Z 715.714,A -85,B 0,C 180,E1 22730.221,E2 22730.221} C_VEL
LIN {X 0,Y 477.642,Z 696.176,A -85,B 0,C 180,E1 22728.494,E2 22728.494} C_VEL
LIN {X 0,Y 470.721,Z 686.264,A -85,B 0,C 180,E1 22727.507,E2 22727.507} C_VEL
LIN {X 0,Y 467.914,Z 682.004,A -85,B 0,C 180,E1 22727.088,E2 22727.088} C_VEL
LIN {X 0,Y 465.654,Z 679.081,A -85,B 0,C 180,E1 22726.756,E2 22726.756} C_VEL
LIN {X 0,Y 465.062,Z 677.192,A -85,B 0,C 180,E1 22726.531,E2 22726.531} C_VEL
LIN {X 0,Y 465.003,Z 676.788,A -85,B 0,C 180,E1 22726.013,E2 22726.013} C_VEL
LIN {X 0,Y 465.002,Z 676.767,A -85,B 0,C 180,E1 22722.298,E2 22722.298} C_VEL
LIN {X 0,Y 465,Z 676.794,A -85,B 0,C 180,E1 22718.693,E2 22718.693} C_VEL
LIN {X 0,Y 465.008,Z 676.792,A -85,B 0,C 180,E1 22714.995,E2 22714.995} C_VEL
LIN {X 0,Y 465.002,Z 676.77,A -85,B 0,C 180,E1 22711.356,E2 22711.356} C_VEL
LIN {X 0,Y 465.007,Z 676.802,A -85,B 0,C 180,E1 22707.643,E2 22707.643} C_VEL
LIN {X 0,Y 465.005,Z 676.801,A -85,B 0,C 180,E1 22703.963,E2 22703.963} C_VEL
LIN {X 0,Y 465.015,Z 676.797,A -85,B 0,C 180,E1 22700.374,E2 22700.374} C_VEL
LIN {X 0,Y 465.014,Z 676.801,A -85,B 0,C 180,E1 22696.617,E2 22696.617} C_VEL
LIN {X 0,Y 465,Z 676.808,A -85,B 0,C 180,E1 22692.922,E2 22692.922} C_VEL
LIN {X 0,Y 465.013,Z 676.812,A -85,B 0,C 180,E1 22689.28,E2 22689.28} C_VEL
LIN {X 0,Y 465.014,Z 676.801,A -85,B 0,C 180,E1 22685.553,E2 22685.553} C_VEL
LIN {X 0,Y 465.004,Z 676.794,A -85,B 0,C 180,E1 22681.849,E2 22681.849} C_VEL
LIN {X 0,Y 465.005,Z 676.802,A -85,B 0,C 180,E1 22678.152,E2 22678.152} C_VEL
LIN {X 0,Y 465.005,Z 676.81,A -85,B 0,C 180,E1 22674.448,E2 22674.448} C_VEL
LIN {X 0,Y 465.013,Z 676.807,A -85,B 0,C 180,E1 22670.845,E2 22670.845} C_VEL
LIN {X 0,Y 464.999,Z 676.78,A -85,B 0,C 180,E1 22667.205,E2 22667.205} C_VEL
LIN {X 0,Y 465.003,Z 676.811,A -85,B 0,C 180,E1 22663.64,E2 22663.64} C_VEL
LIN {X 0,Y 465.007,Z 676.788,A -85,B 0,C 180,E1 22659.878,E2 22659.878} C_VEL
LIN {X 0,Y 465,Z 676.794,A -85,B 0,C 180,E1 22656.291,E2 22656.291} C_VEL
LIN {X 0,Y 465.014,Z 676.81,A -85,B 0,C 180,E1 22652.604,E2 22652.604} C_VEL
LIN {X 0,Y 465.001,Z 676.805,A -85,B 0,C 180,E1 22648.932,E2 22648.932} C_VEL
LIN {X 0,Y 465.008,Z 676.795,A -85,B 0,C 180,E1 22645.22,E2 22645.22} C_VEL
LIN {X 0,Y 465.006,Z 676.797,A -85,B 0,C 180,E1 22641.504,E2 22641.504} C_VEL
LIN {X 0,Y 465.054,Z 677.159,A -85,B 0,C 180,E1 22640.223,E2 22640.223} C_VEL
LIN {X 0,Y 466.602,Z 680.683,A -85,B 0,C 180,E1 22639.674,E2 22639.674} C_VEL
LIN {X 0,Y 474.843,Z 697.679,A -85,B 0,C 180,E1 22637.229,E2 22637.229} C_VEL
LIN {X 0,Y 483.668,Z 717.716,A -85,B 0,C 180,E1 22634.655,E2 22634.655} C_VEL
LIN {X 0,Y 486.687,Z 725.084,A -85,B 0,C 180,E1 22633.779,E2 22633.779} C_VEL
LIN {X 0,Y 485.308,Z 748.503,A -85,B 0,C 180,E1 22632.108,E2 22632.108} C_VEL
LIN {X 0,Y 490.687,Z 786.143,A -85,B 0,C 180,E1 22630.857,E2 22630.857} C_VEL
LIN {X 0,Y 486.12,Z 1017.142,A -85,B 0,C 180,E1 22627.065,E2 22627.065} C_VEL
LIN {X 0,Y 485.075,Z 1061.693,A -85,B 0,C 180,E1 22626.308,E2 22626.308} C_VEL
LIN {X 0,Y 483.864,Z 1083.559,A -85,B 0,C 180,E1 22625.739,E2 22625.739} C_VEL
LIN {X 0,Y 482.36,Z 1105.102,A -85,B 0,C 180,E1 22624.968,E2 22624.968} C_VEL
LIN {X 0,Y 480.676,Z 1125.851,A -85,B 0,C 180,E1 22624.023,E2 22624.023} C_VEL
LIN {X 0,Y 478.747,Z 1146.933,A -85,B 0,C 180,E1 22622.816,E2 22622.816} C_VEL
LIN {X 0,Y 476.693,Z 1167.638,A -85,B 0,C 180,E1 22621.386,E2 22621.386} C_VEL
LIN {X 0,Y 474.713,Z 1187.073,A -85,B 0,C 180,E1 22619.8,E2 22619.8} C_VEL
LIN {X 0,Y 472.729,Z 1205.819,A -85,B 0,C 180,E1 22618.004,E2 22618.004} C_VEL
LIN {X 0,Y 470.932,Z 1222.895,A -85,B 0,C 180,E1 22616.092,E2 22616.092} C_VEL
LIN {X 0,Y 469.394,Z 1236.563,A -85,B 0,C 180,E1 22614.261,E2 22614.261} C_VEL
LIN {X 0,Y 467.846,Z 1250.322,A -85,B 0,C 180,E1 22612.094,E2 22612.094} C_VEL
LIN {X 0,Y 466.509,Z 1263.546,A -85,B 0,C 180,E1 22609.663,E2 22609.663} C_VEL
LIN {X 0,Y 465.528,Z 1274.749,A -85,B 0,C 180,E1 22607.241,E2 22607.241} C_VEL
LIN {X 0,Y 464.811,Z 1284.512,A -85,B 0,C 180,E1 22604.704,E2 22604.704} C_VEL
LIN {X 0,Y 464.35,Z 1292.533,A -85,B 0,C 180,E1 22602.159,E2 22602.159} C_VEL
LIN {X 0,Y 464.087,Z 1299.129,A -85,B 0,C 180,E1 22599.549,E2 22599.549} C_VEL
LIN {X 0,Y 463.965,Z 1303.813,A -85,B 0,C 180,E1 22597.056,E2 22597.056} C_VEL
LIN {X 0,Y 463.914,Z 1307.332,A -85,B 0,C 180,E1 22594.326,E2 22594.326} C_VEL
LIN {X 0,Y 463.899,Z 1309.085,A -85,B 0,C 180,E1 22591.853,E2 22591.853} C_VEL
LIN {X 0,Y 463.898,Z 1309.371,A -85,B 0,C 180,E1 22589.259,E2 22589.259} C_VEL
LIN {X 0,Y 463.912,Z 1308.235,A -85,B 0,C 180,E1 22586.664,E2 22586.664} C_VEL
LIN {X 0,Y 463.93,Z 1305.457,A -85,B 0,C 180,E1 22584.062,E2 22584.062} C_VEL
LIN {X 0,Y 464.026,Z 1300.907,A -85,B 0,C 180,E1 22581.325,E2 22581.325} C_VEL
LIN {X 0,Y 464.246,Z 1294.937,A -85,B 0,C 180,E1 22578.698,E2 22578.698} C_VEL
LIN {X 0,Y 464.627,Z 1287.476,A -85,B 0,C 180,E1 22576.181,E2 22576.181} C_VEL
LIN {X 0,Y 465.279,Z 1277.837,A -85,B 0,C 180,E1 22573.522,E2 22573.522} C_VEL
LIN {X 0,Y 466.199,Z 1267.095,A -85,B 0,C 180,E1 22571.051,E2 22571.051} C_VEL
LIN {X 0,Y 467.389,Z 1254.758,A -85,B 0,C 180,E1 22568.675,E2 22568.675} C_VEL
LIN {X 0,Y 468.906,Z 1240.711,A -85,B 0,C 180,E1 22566.368,E2 22566.368} C_VEL
LIN {X 0,Y 470.625,Z 1225.783,A -85,B 0,C 180,E1 22564.263,E2 22564.263} C_VEL
LIN {X 0,Y 472.212,Z 1210.74,A -85,B 0,C 180,E1 22562.521,E2 22562.521} C_VEL
LIN {X 0,Y 474.137,Z 1192.236,A -85,B 0,C 180,E1 22560.671,E2 22560.671} C_VEL
LIN {X 0,Y 476.158,Z 1173.255,A -85,B 0,C 180,E1 22559.04,E2 22559.04} C_VEL
LIN {X 0,Y 478.055,Z 1153.815,A -85,B 0,C 180,E1 22557.628,E2 22557.628} C_VEL
LIN {X 0,Y 480.058,Z 1132.862,A -85,B 0,C 180,E1 22556.358,E2 22556.358} C_VEL
LIN {X 0,Y 481.844,Z 1111.865,A -85,B 0,C 180,E1 22555.311,E2 22555.311} C_VEL
LIN {X 0,Y 483.421,Z 1090.362,A -85,B 0,C 180,E1 22554.479,E2 22554.479} C_VEL
LIN {X 0,Y 484.758,Z 1067.92,A -85,B 0,C 180,E1 22553.838,E2 22553.838} C_VEL
LIN {X 0,Y 485.615,Z 1044.176,A -85,B 0,C 180,E1 22553.373,E2 22553.373} C_VEL
LIN {X 0,Y 489.938,Z 821.828,A -85,B 0,C 180,E1 22549.733,E2 22549.733} C_VEL
LIN {X 0,Y 490.537,Z 783.876,A -85,B 0,C 180,E1 22549.086,E2 22549.086} C_VEL
LIN {X 0,Y 485.258,Z 747.487,A -85,B 0,C 180,E1 22547.842,E2 22547.842} C_VEL
LIN {X 0,Y 486.517,Z 724.568,A -85,B 0,C 180,E1 22546.166,E2 22546.166} C_VEL
LIN {X 0,Y 477.475,Z 703.447,A -85,B 0,C 180,E1 22543.546,E2 22543.546} C_VEL
LIN {X 0,Y 469.023,Z 685.33,A -85,B 0,C 180,E1 22541.04,E2 22541.04} C_VEL
LIN {X 0,Y 465.096,Z 677.388,A -85,B 0,C 180,E1 22539.822,E2 22539.822} C_VEL
LIN {X 0,Y 465.016,Z 676.833,A -85,B 0,C 180,E1 22539.477,E2 22539.477} C_VEL
LIN {X 0,Y 465.004,Z 676.814,A -85,B 0,C 180,E1 22535.793,E2 22535.793} C_VEL
LIN {X 0,Y 465.007,Z 676.813,A -85,B 0,C 180,E1 22532.079,E2 22532.079} C_VEL
LIN {X 0,Y 465.009,Z 676.796,A -85,B 0,C 180,E1 22528.372,E2 22528.372} C_VEL
LIN {X 0,Y 464.999,Z 676.786,A -85,B 0,C 180,E1 22524.654,E2 22524.654} C_VEL
LIN {X 0,Y 465.013,Z 676.806,A -85,B 0,C 180,E1 22521.043,E2 22521.043} C_VEL
LIN {X 0,Y 465,Z 676.806,A -85,B 0,C 180,E1 22517.317,E2 22517.317} C_VEL
LIN {X 0,Y 465.005,Z 676.783,A -85,B 0,C 180,E1 22513.681,E2 22513.681} C_VEL
LIN {X 0,Y 465.005,Z 676.81,A -85,B 0,C 180,E1 22510.014,E2 22510.014} C_VEL
LIN {X 0,Y 465,Z 676.807,A -85,B 0,C 180,E1 22506.42,E2 22506.42} C_VEL
LIN {X 0,Y 465.011,Z 676.797,A -85,B 0,C 180,E1 22502.711,E2 22502.711} C_VEL
LIN {X 0,Y 465.005,Z 676.805,A -85,B 0,C 180,E1 22499.137,E2 22499.137} C_VEL
LIN {X 0,Y 465.003,Z 676.81,A -85,B 0,C 180,E1 22495.437,E2 22495.437} C_VEL
LIN {X 0,Y 465.009,Z 676.809,A -85,B 0,C 180,E1 22491.717,E2 22491.717} C_VEL
LIN {X 0,Y 465.014,Z 676.799,A -85,B 0,C 180,E1 22488.041,E2 22488.041} C_VEL
LIN {X 0,Y 465.012,Z 676.799,A -85,B 0,C 180,E1 22484.409,E2 22484.409} C_VEL
LIN {X 0,Y 465.001,Z 676.806,A -85,B 0,C 180,E1 22480.662,E2 22480.662} C_VEL
LIN {X 0,Y 465.017,Z 676.805,A -85,B 0,C 180,E1 22476.961,E2 22476.961} C_VEL
LIN {X 0,Y 465.013,Z 676.81,A -85,B 0,C 180,E1 22473.295,E2 22473.295} C_VEL
LIN {X 0,Y 464.996,Z 676.757,A -85,B 0,C 180,E1 22469.648,E2 22469.648} C_VEL
LIN {X 0,Y 465.011,Z 676.81,A -85,B 0,C 180,E1 22466.01,E2 22466.01} C_VEL
LIN {X 0,Y 464.999,Z 676.77,A -85,B 0,C 180,E1 22462.304,E2 22462.304} C_VEL
LIN {X 0,Y 465.006,Z 676.783,A -85,B 0,C 180,E1 22458.691,E2 22458.691} C_VEL
LIN {X 0,Y 465.007,Z 676.814,A -85,B 0,C 180,E1 22454.975,E2 22454.975} C_VEL
LIN {X 0,Y 465.03,Z 676.994,A -85,B 0,C 180,E1 22453.432,E2 22453.432} C_VEL
LIN {X 0,Y 465.436,Z 678.547,A -85,B 0,C 180,E1 22453.193,E2 22453.193} C_VEL
LIN {X 0,Y 467.401,Z 681.553,A -85,B 0,C 180,E1 22452.889,E2 22452.889} C_VEL
LIN {X 0,Y 468.621,Z 682.972,A -85,B 0,C 180,E1 22452.715,E2 22452.715} C_VEL
LIN {X 0,Y 471.45,Z 687.063,A -85,B 0,C 180,E1 22452.299,E2 22452.299} C_VEL
LIN {X 0,Y 486.658,Z 709.831,A -85,B 0,C 180,E1 22450.179,E2 22450.179} C_VEL
LIN {X 0,Y 490.365,Z 716.064,A -85,B 0,C 180,E1 22449.679,E2 22449.679} C_VEL
LIN {X 0,Y 487.913,Z 827.764,A -85,B 0,C 180,E1 22447.822,E2 22447.822} C_VEL
LIN {X 0,Y 486.999,Z 835.458,A -85,B 0,C 180,E1 22447.767,E2 22447.767} C_VEL
LIN {X 0,Y 481.67,Z 856.006,A -85,B 0,C 180,E1 22447.895,E2 22447.895} C_VEL
LIN {X 0,Y 480.93,Z 862.612,A -85,B 0,C 180,E1 22447.842,E2 22447.842} C_VEL
LIN {X 0,Y 479.492,Z 923.785,A -85,B 0,C 180,E1 22446.787,E2 22446.787} C_VEL
LIN {X 0,Y 478.428,Z 945.193,A -85,B 0,C 180,E1 22446.199,E2 22446.199} C_VEL
LIN {X 0,Y 477.038,Z 965.892,A -85,B 0,C 180,E1 22445.417,E2 22445.417} C_VEL
LIN {X 0,Y 475.382,Z 985.676,A -85,B 0,C 180,E1 22444.455,E2 22444.455} C_VEL
LIN {X 0,Y 473.385,Z 1004.528,A -85,B 0,C 180,E1 22443.308,E2 22443.308} C_VEL
LIN {X 0,Y 471.017,Z 1024.433,A -85,B 0,C 180,E1 22441.836,E2 22441.836} C_VEL
LIN {X 0,Y 468.75,Z 1041.841,A -85,B 0,C 180,E1 22440.295,E2 22440.295} C_VEL
LIN {X 0,Y 466.397,Z 1058.299,A -85,B 0,C 180,E1 22438.558,E2 22438.558} C_VEL
LIN {X 0,Y 464.096,Z 1074.011,A -85,B 0,C 180,E1 22436.609,E2 22436.609} C_VEL
LIN {X 0,Y 462.032,Z 1088.207,A -85,B 0,C 180,E1 22434.55,E2 22434.55} C_VEL
LIN {X 0,Y 460.19,Z 1101.057,A -85,B 0,C 180,E1 22432.347,E2 22432.347} C_VEL
LIN {X 0,Y 458.59,Z 1115.237,A -85,B 0,C 180,E1 22429.618,E2 22429.618} C_VEL
LIN {X 0,Y 457.512,Z 1126.635,A -85,B 0,C 180,E1 22427.028,E2 22427.028} C_VEL
LIN {X 0,Y 456.787,Z 1136.124,A -85,B 0,C 180,E1 22424.449,E2 22424.449} C_VEL
LIN {X 0,Y 456.329,Z 1143.758,A -85,B 0,C 180,E1 22421.885,E2 22421.885} C_VEL
LIN {X 0,Y 456.074,Z 1150.057,A -85,B 0,C 180,E1 22419.209,E2 22419.209} C_VEL
LIN {X 0,Y 455.957,Z 1154.76,A -85,B 0,C 180,E1 22416.547,E2 22416.547} C_VEL
LIN {X 0,Y 455.903,Z 1157.746,A -85,B 0,C 180,E1 22413.898,E2 22413.898} C_VEL
LIN {X 0,Y 455.907,Z 1159.295,A -85,B 0,C 180,E1 22411.131,E2 22411.131} C_VEL
LIN {X 0,Y 455.906,Z 1159.266,A -85,B 0,C 180,E1 22408.618,E2 22408.618} C_VEL
LIN {X 0,Y 455.909,Z 1157.714,A -85,B 0,C 180,E1 22405.976,E2 22405.976} C_VEL
LIN {X 0,Y 455.963,Z 1154.708,A -85,B 0,C 180,E1 22403.326,E2 22403.326} C_VEL
LIN {X 0,Y 456.074,Z 1149.981,A -85,B 0,C 180,E1 22400.664,E2 22400.664} C_VEL
LIN {X 0,Y 456.352,Z 1143.298,A -85,B 0,C 180,E1 22397.858,E2 22397.858} C_VEL
LIN {X 0,Y 456.829,Z 1135.583,A -85,B 0,C 180,E1 22395.293,E2 22395.293} C_VEL
LIN {X 0,Y 457.574,Z 1125.958,A -85,B 0,C 180,E1 22392.712,E2 22392.712} C_VEL
LIN {X 0,Y 458.672,Z 1114.396,A -85,B 0,C 180,E1 22390.12,E2 22390.12} C_VEL
LIN {X 0,Y 460.617,Z 1097.949,A -85,B 0,C 180,E1 22387.001,E2 22387.001} C_VEL
LIN {X 0,Y 462.692,Z 1083.638,A -85,B 0,C 180,E1 22384.668,E2 22384.668} C_VEL
LIN {X 0,Y 464.895,Z 1068.675,A -85,B 0,C 180,E1 22382.597,E2 22382.597} C_VEL
LIN {X 0,Y 467.218,Z 1052.689,A -85,B 0,C 180,E1 22380.726,E2 22380.726} C_VEL
LIN {X 0,Y 469.54,Z 1035.781,A -85,B 0,C 180,E1 22379.053,E2 22379.053} C_VEL
LIN {X 0,Y 471.916,Z 1017.262,A -85,B 0,C 180,E1 22377.508,E2 22377.508} C_VEL
LIN {X 0,Y 474.029,Z 998.939,A -85,B 0,C 180,E1 22376.236,E2 22376.236} C_VEL
LIN {X 0,Y 475.874,Z 979.745,A -85,B 0,C 180,E1 22375.146,E2 22375.146} C_VEL
LIN {X 0,Y 477.571,Z 958.814,A -85,B 0,C 180,E1 22374.2,E2 22374.2} C_VEL
LIN {X 0,Y 478.829,Z 938.671,A -85,B 0,C 180,E1 22373.51,E2 22373.51} C_VEL
LIN {X 0,Y 479.656,Z 917.301,A -85,B 0,C 180,E1 22372.993,E2 22372.993} C_VEL
LIN {X 0,Y 484.259,Z 719.086,A -85,B 0,C 180,E1 22369.659,E2 22369.659} C_VEL
LIN {X 0,Y 471.912,Z 700.272,A -85,B 0,C 180,E1 22367.932,E2 22367.932} C_VEL
LIN {X 0,Y 463.151,Z 687.628,A -85,B 0,C 180,E1 22366.634,E2 22366.634} C_VEL
LIN {X 0,Y 459.994,Z 683.027,A -85,B 0,C 180,E1 22366.146,E2 22366.146} C_VEL
LIN {X 0,Y 457.771,Z 680.198,A -85,B 0,C 180,E1 22365.804,E2 22365.804} C_VEL
LIN {X 0,Y 457.15,Z 678.28,A -85,B 0,C 180,E1 22365.584,E2 22365.584} C_VEL
LIN {X 0,Y 457.069,Z 677.8,A -85,B 0,C 180,E1 22365.222,E2 22365.222} C_VEL
LIN {X 0,Y 457.072,Z 677.762,A -85,B 0,C 180,E1 22361.516,E2 22361.516} C_VEL
LIN {X 0,Y 457.059,Z 677.759,A -85,B 0,C 180,E1 22357.843,E2 22357.843} C_VEL
LIN {X 0,Y 457.066,Z 677.8,A -85,B 0,C 180,E1 22354.208,E2 22354.208} C_VEL
LIN {X 0,Y 457.061,Z 677.744,A -85,B 0,C 180,E1 22350.472,E2 22350.472} C_VEL
LIN {X 0,Y 457.071,Z 677.797,A -85,B 0,C 180,E1 22346.784,E2 22346.784} C_VEL
LIN {X 0,Y 457.077,Z 677.793,A -85,B 0,C 180,E1 22343.052,E2 22343.052} C_VEL
LIN {X 0,Y 457.063,Z 677.793,A -85,B 0,C 180,E1 22339.421,E2 22339.421} C_VEL
LIN {X 0,Y 457.075,Z 677.786,A -85,B 0,C 180,E1 22335.739,E2 22335.739} C_VEL
LIN {X 0,Y 457.075,Z 677.788,A -85,B 0,C 180,E1 22331.994,E2 22331.994} C_VEL
LIN {X 0,Y 457.069,Z 677.798,A -85,B 0,C 180,E1 22328.301,E2 22328.301} C_VEL
LIN {X 0,Y 457.064,Z 677.799,A -85,B 0,C 180,E1 22324.517,E2 22324.517} C_VEL
LIN {X 0,Y 457.069,Z 677.795,A -85,B 0,C 180,E1 22320.752,E2 22320.752} C_VEL
LIN {X 0,Y 457.071,Z 677.785,A -85,B 0,C 180,E1 22316.991,E2 22316.991} C_VEL
LIN {X 0,Y 457.066,Z 677.791,A -85,B 0,C 180,E1 22313.276,E2 22313.276} C_VEL
LIN {X 0,Y 457.067,Z 677.797,A -85,B 0,C 180,E1 22309.539,E2 22309.539} C_VEL
LIN {X 0,Y 457.061,Z 677.778,A -85,B 0,C 180,E1 22305.818,E2 22305.818} C_VEL
LIN {X 0,Y 457.069,Z 677.779,A -85,B 0,C 180,E1 22302.092,E2 22302.092} C_VEL
LIN {X 0,Y 457.062,Z 677.799,A -85,B 0,C 180,E1 22298.387,E2 22298.387} C_VEL
LIN {X 0,Y 457.067,Z 677.776,A -85,B 0,C 180,E1 22294.75,E2 22294.75} C_VEL
LIN {X 0,Y 457.062,Z 677.776,A -85,B 0,C 180,E1 22291.045,E2 22291.045} C_VEL
LIN {X 0,Y 457.066,Z 677.79,A -85,B 0,C 180,E1 22287.371,E2 22287.371} C_VEL
LIN {X 0,Y 457.066,Z 677.794,A -85,B 0,C 180,E1 22283.61,E2 22283.61} C_VEL
LIN {X 0,Y 457.098,Z 678.033,A -85,B 0,C 180,E1 22281.171,E2 22281.171} C_VEL
LIN {X 0,Y 458.499,Z 681.455,A -85,B 0,C 180,E1 22280.611,E2 22280.611} C_VEL
LIN {X 0,Y 465.264,Z 694.901,A -85,B 0,C 180,E1 22278.556,E2 22278.556} C_VEL
LIN {X 0,Y 473.88,Z 713.941,A -85,B 0,C 180,E1 22275.955,E2 22275.955} C_VEL
LIN {X 0,Y 479.943,Z 728.714,A -85,B 0,C 180,E1 22274.132,E2 22274.132} C_VEL
LIN {X 0,Y 478.803,Z 747.003,A -85,B 0,C 180,E1 22272.815,E2 22272.815} C_VEL
LIN {X 0,Y 484.502,Z 787.593,A -85,B 0,C 180,E1 22271.438,E2 22271.438} C_VEL
LIN {X 0,Y 479.628,Z 1017.895,A -85,B 0,C 180,E1 22267.613,E2 22267.613} C_VEL
LIN {X 0,Y 478.559,Z 1060.389,A -85,B 0,C 180,E1 22266.88,E2 22266.88} C_VEL
LIN {X 0,Y 477.233,Z 1082.431,A -85,B 0,C 180,E1 22266.303,E2 22266.303} C_VEL
LIN {X 0,Y 475.586,Z 1104.332,A -85,B 0,C 180,E1 22265.508,E2 22265.508} C_VEL
LIN {X 0,Y 473.713,Z 1125.555,A -85,B 0,C 180,E1 22264.521,E2 22264.521} C_VEL
LIN {X 0,Y 471.657,Z 1146.502,A -85,B 0,C 180,E1 22263.301,E2 22263.301} C_VEL
LIN {X 0,Y 469.49,Z 1166.678,A -85,B 0,C 180,E1 22261.88,E2 22261.88} C_VEL
LIN {X 0,Y 467.336,Z 1186.231,A -85,B 0,C 180,E1 22260.254,E2 22260.254} C_VEL
LIN {X 0,Y 465.215,Z 1204.969,A -85,B 0,C 180,E1 22258.427,E2 22258.427} C_VEL
LIN {X 0,Y 463.286,Z 1222.146,A -85,B 0,C 180,E1 22256.465,E2 22256.465} C_VEL
LIN {X 0,Y 461.399,Z 1239.464,A -85,B 0,C 180,E1 22254.174,E2 22254.174} C_VEL
LIN {X 0,Y 460.293,Z 1249.594,A -85,B 0,C 180,E1 22252.603,E2 22252.603} C_VEL
LIN {X 0,Y 458.792,Z 1263.256,A -85,B 0,C 180,E1 22250.068,E2 22250.068} C_VEL
LIN {X 0,Y 457.746,Z 1274.231,A -85,B 0,C 180,E1 22247.675,E2 22247.675} C_VEL
LIN {X 0,Y 456.938,Z 1284.052,A -85,B 0,C 180,E1 22245.093,E2 22245.093} C_VEL
LIN {X 0,Y 456.402,Z 1292.469,A -85,B 0,C 180,E1 22242.397,E2 22242.397} C_VEL
LIN {X 0,Y 456.106,Z 1299.129,A -85,B 0,C 180,E1 22239.718,E2 22239.718} C_VEL
LIN {X 0,Y 455.967,Z 1304.019,A -85,B 0,C 180,E1 22237.053,E2 22237.053} C_VEL
LIN {X 0,Y 455.912,Z 1307.445,A -85,B 0,C 180,E1 22234.276,E2 22234.276} C_VEL
LIN {X 0,Y 455.896,Z 1309.209,A -85,B 0,C 180,E1 22231.634,E2 22231.634} C_VEL
LIN {X 0,Y 455.903,Z 1309.348,A -85,B 0,C 180,E1 22229.12,E2 22229.12} C_VEL
LIN {X 0,Y 455.909,Z 1308.123,A -85,B 0,C 180,E1 22226.48,E2 22226.48} C_VEL
LIN {X 0,Y 455.93,Z 1305.457,A -85,B 0,C 180,E1 22223.958,E2 22223.958} C_VEL
LIN {X 0,Y 456.043,Z 1300.907,A -85,B 0,C 180,E1 22221.172,E2 22221.172} C_VEL
LIN {X 0,Y 456.283,Z 1294.937,A -85,B 0,C 180,E1 22218.498,E2 22218.498} C_VEL
LIN {X 0,Y 456.706,Z 1287.343,A -85,B 0,C 180,E1 22215.894,E2 22215.894} C_VEL
LIN {X 0,Y 457.413,Z 1277.794,A -85,B 0,C 180,E1 22213.219,E2 22213.219} C_VEL
LIN {X 0,Y 458.391,Z 1267.353,A -85,B 0,C 180,E1 22210.77,E2 22210.77} C_VEL
LIN {X 0,Y 459.713,Z 1254.757,A -85,B 0,C 180,E1 22208.301,E2 22208.301} C_VEL
LIN {X 0,Y 461.026,Z 1243.053,A -85,B 0,C 180,E1 22206.346,E2 22206.346} C_VEL
LIN {X 0,Y 462.714,Z 1227.427,A -85,B 0,C 180,E1 22204.189,E2 22204.189} C_VEL
LIN {X 0,Y 464.61,Z 1210.338,A -85,B 0,C 180,E1 22202.162,E2 22202.162} C_VEL
LIN {X 0,Y 466.767,Z 1191.15,A -85,B 0,C 180,E1 22200.202,E2 22200.202} C_VEL
LIN {X 0,Y 468.961,Z 1171.77,A -85,B 0,C 180,E1 22198.511,E2 22198.511} C_VEL
LIN {X 0,Y 471.021,Z 1152.341,A -85,B 0,C 180,E1 22197.084,E2 22197.084} C_VEL
LIN {X 0,Y 473.212,Z 1130.752,A -85,B 0,C 180,E1 22195.764,E2 22195.764} C_VEL
LIN {X 0,Y 475.091,Z 1110.346,A -85,B 0,C 180,E1 22194.742,E2 22194.742} C_VEL
LIN {X 0,Y 476.772,Z 1089.17,A -85,B 0,C 180,E1 22193.917,E2 22193.917} C_VEL
LIN {X 0,Y 478.218,Z 1066.486,A -85,B 0,C 180,E1 22193.263,E2 22193.263} C_VEL
LIN {X 0,Y 479.134,Z 1042.629,A -85,B 0,C 180,E1 22192.793,E2 22192.793} C_VEL
LIN {X 0,Y 483.769,Z 820.14,A -85,B 0,C 180,E1 22189.106,E2 22189.106} C_VEL
LIN {X 0,Y 484.375,Z 785.459,A -85,B 0,C 180,E1 22188.509,E2 22188.509} C_VEL
LIN {X 0,Y 478.746,Z 746.096,A -85,B 0,C 180,E1 22187.143,E2 22187.143} C_VEL
LIN {X 0,Y 479.921,Z 728.401,A -85,B 0,C 180,E1 22185.842,E2 22185.842} C_VEL
LIN {X 0,Y 471.252,Z 707.935,A -85,B 0,C 180,E1 22183.26,E2 22183.26} C_VEL
LIN {X 0,Y 462.833,Z 690.002,A -85,B 0,C 180,E1 22180.723,E2 22180.723} C_VEL
LIN {X 0,Y 458.48,Z 681.431,A -85,B 0,C 180,E1 22179.391,E2 22179.391} C_VEL
LIN {X 0,Y 457.093,Z 678.022,A -85,B 0,C 180,E1 22178.814,E2 22178.814} C_VEL
LIN {X 0,Y 457.064,Z 677.793,A -85,B 0,C 180,E1 22175.276,E2 22175.276} C_VEL
LIN {X 0,Y 457.067,Z 677.802,A -85,B 0,C 180,E1 22171.522,E2 22171.522} C_VEL
LIN {X 0,Y 457.064,Z 677.796,A -85,B 0,C 180,E1 22167.902,E2 22167.902} C_VEL
LIN {X 0,Y 457.068,Z 677.775,A -85,B 0,C 180,E1 22164.146,E2 22164.146} C_VEL
LIN {X 0,Y 457.061,Z 677.784,A -85,B 0,C 180,E1 22160.488,E2 22160.488} C_VEL
LIN {X 0,Y 457.07,Z 677.797,A -85,B 0,C 180,E1 22156.783,E2 22156.783} C_VEL
LIN {X 0,Y 457.063,Z 677.767,A -85,B 0,C 180,E1 22153.15,E2 22153.15} C_VEL
LIN {X 0,Y 457.072,Z 677.801,A -85,B 0,C 180,E1 22149.409,E2 22149.409} C_VEL
LIN {X 0,Y 457.067,Z 677.797,A -85,B 0,C 180,E1 22145.649,E2 22145.649} C_VEL
LIN {X 0,Y 457.062,Z 677.791,A -85,B 0,C 180,E1 22142.006,E2 22142.006} C_VEL
LIN {X 0,Y 457.068,Z 677.782,A -85,B 0,C 180,E1 22138.245,E2 22138.245} C_VEL
LIN {X 0,Y 457.072,Z 677.793,A -85,B 0,C 180,E1 22134.602,E2 22134.602} C_VEL
LIN {X 0,Y 457.07,Z 677.799,A -85,B 0,C 180,E1 22130.938,E2 22130.938} C_VEL
LIN {X 0,Y 457.063,Z 677.797,A -85,B 0,C 180,E1 22127.235,E2 22127.235} C_VEL
LIN {X 0,Y 457.075,Z 677.787,A -85,B 0,C 180,E1 22123.609,E2 22123.609} C_VEL
LIN {X 0,Y 457.077,Z 677.786,A -85,B 0,C 180,E1 22119.913,E2 22119.913} C_VEL
LIN {X 0,Y 457.063,Z 677.792,A -85,B 0,C 180,E1 22116.264,E2 22116.264} C_VEL
LIN {X 0,Y 457.075,Z 677.791,A -85,B 0,C 180,E1 22112.512,E2 22112.512} C_VEL
LIN {X 0,Y 457.066,Z 677.752,A -85,B 0,C 180,E1 22108.771,E2 22108.771} C_VEL
LIN {X 0,Y 457.069,Z 677.783,A -85,B 0,C 180,E1 22105.115,E2 22105.115} C_VEL
LIN {X 0,Y 457.06,Z 677.776,A -85,B 0,C 180,E1 22101.347,E2 22101.347} C_VEL
LIN {X 0,Y 457.06,Z 677.756,A -85,B 0,C 180,E1 22097.81,E2 22097.81} C_VEL
LIN {X 0,Y 457.09,Z 677.937,A -85,B 0,C 180,E1 22094.424,E2 22094.424} C_VEL
LIN {X 0,Y 457.418,Z 679.321,A -85,B 0,C 180,E1 22094.173,E2 22094.173} C_VEL
LIN {X 0,Y 459.322,Z 682.424,A -85,B 0,C 180,E1 22093.857,E2 22093.857} C_VEL
LIN {X 0,Y 460.777,Z 684.031,A -85,B 0,C 180,E1 22093.641,E2 22093.641} C_VEL
LIN {X 0,Y 463.465,Z 687.966,A -85,B 0,C 180,E1 22093.227,E2 22093.227} C_VEL
LIN {X 0,Y 476.974,Z 707.758,A -85,B 0,C 180,E1 22091.256,E2 22091.256} C_VEL
LIN {X 0,Y 484.256,Z 719.361,A -85,B 0,C 180,E1 22090.245,E2 22090.245} C_VEL
LIN {X 0,Y 480.93,Z 862.612,A -85,B 0,C 180,E1 22087.842,E2 22087.842} C_VEL
LIN {X 0,Y 479.992,Z 870.304,A -85,B 0,C 180,E1 22087.788,E2 22087.788} C_VEL
LIN {X 0,Y 474.682,Z 890.846,A -85,B 0,C 180,E1 22087.916,E2 22087.916} C_VEL
LIN {X 0,Y 473.902,Z 897.452,A -85,B 0,C 180,E1 22087.866,E2 22087.866} C_VEL
LIN {X 0,Y 473.043,Z 927.861,A -85,B 0,C 180,E1 22087.297,E2 22087.297} C_VEL
LIN {X 0,Y 471.958,Z 948.958,A -85,B 0,C 180,E1 22086.689,E2 22086.689} C_VEL
LIN {X 0,Y 470.527,Z 968.737,A -85,B 0,C 180,E1 22085.907,E2 22085.907} C_VEL
LIN {X 0,Y 468.789,Z 988.213,A -85,B 0,C 180,E1 22084.935,E2 22084.935} C_VEL
LIN {X 0,Y 466.707,Z 1006.912,A -85,B 0,C 180,E1 22083.774,E2 22083.774} C_VEL
LIN {X 0,Y 464.333,Z 1025.834,A -85,B 0,C 180,E1 22082.35,E2 22082.35} C_VEL
LIN {X 0,Y 461.886,Z 1043.619,A -85,B 0,C 180,E1 22080.751,E2 22080.751} C_VEL
LIN {X 0,Y 459.363,Z 1060.365,A -85,B 0,C 180,E1 22078.955,E2 22078.955} C_VEL
LIN {X 0,Y 456.957,Z 1075.801,A -85,B 0,C 180,E1 22077.001,E2 22077.001} C_VEL
LIN {X 0,Y 454.816,Z 1089.615,A -85,B 0,C 180,E1 22074.966,E2 22074.966} C_VEL
LIN {X 0,Y 452.839,Z 1102.467,A -85,B 0,C 180,E1 22072.73,E2 22072.73} C_VEL
LIN {X 0,Y 451.156,Z 1114.04,A -85,B 0,C 180,E1 22070.361,E2 22070.361} C_VEL
LIN {X 0,Y 449.484,Z 1128.695,A -85,B 0,C 180,E1 22066.808,E2 22066.808} C_VEL
LIN {X 0,Y 448.755,Z 1137.745,A -85,B 0,C 180,E1 22064.187,E2 22064.187} C_VEL
LIN {X 0,Y 448.311,Z 1145.146,A -85,B 0,C 180,E1 22061.579,E2 22061.579} C_VEL
LIN {X 0,Y 448.067,Z 1150.822,A -85,B 0,C 180,E1 22058.986,E2 22058.986} C_VEL
LIN {X 0,Y 447.938,Z 1155.404,A -85,B 0,C 180,E1 22056.15,E2 22056.15} C_VEL
LIN {X 0,Y 447.906,Z 1158.088,A -85,B 0,C 180,E1 22053.583,E2 22053.583} C_VEL
LIN {X 0,Y 447.904,Z 1159.34,A -85,B 0,C 180,E1 22050.895,E2 22050.895} C_VEL
LIN {X 0,Y 447.899,Z 1159.177,A -85,B 0,C 180,E1 22048.209,E2 22048.209} C_VEL
LIN {X 0,Y 447.918,Z 1157.372,A -85,B 0,C 180,E1 22045.519,E2 22045.519} C_VEL
LIN {X 0,Y 447.967,Z 1153.884,A -85,B 0,C 180,E1 22042.691,E2 22042.691} C_VEL
LIN {X 0,Y 448.119,Z 1149.216,A -85,B 0,C 180,E1 22040.108,E2 22040.108} C_VEL
LIN {X 0,Y 448.423,Z 1142.942,A -85,B 0,C 180,E1 22037.51,E2 22037.51} C_VEL
LIN {X 0,Y 448.961,Z 1135.13,A -85,B 0,C 180,E1 22034.897,E2 22034.897} C_VEL
LIN {X 0,Y 449.794,Z 1125.438,A -85,B 0,C 180,E1 22032.27,E2 22032.27} C_VEL
LIN {X 0,Y 451.393,Z 1112.432,A -85,B 0,C 180,E1 22029.189,E2 22029.189} C_VEL
LIN {X 0,Y 453.083,Z 1100.788,A -85,B 0,C 180,E1 22026.871,E2 22026.871} C_VEL
LIN {X 0,Y 455.124,Z 1087.645,A -85,B 0,C 180,E1 22024.635,E2 22024.635} C_VEL
LIN {X 0,Y 457.448,Z 1072.802,A -85,B 0,C 180,E1 22022.498,E2 22022.498} C_VEL
LIN {X 0,Y 459.874,Z 1056.977,A -85,B 0,C 180,E1 22020.57,E2 22020.57} C_VEL
LIN {X 0,Y 462.493,Z 1039.268,A -85,B 0,C 180,E1 22018.746,E2 22018.746} C_VEL
LIN {X 0,Y 464.957,Z 1021.316,A -85,B 0,C 180,E1 22017.188,E2 22017.188} C_VEL
LIN {X 0,Y 467.147,Z 1003.236,A -85,B 0,C 180,E1 22015.892,E2 22015.892} C_VEL
LIN {X 0,Y 469.264,Z 982.944,A -85,B 0,C 180,E1 22014.692,E2 22014.692} C_VEL
LIN {X 0,Y 471.035,Z 962.513,A -85,B 0,C 180,E1 22013.728,E2 22013.728} C_VEL
LIN {X 0,Y 472.379,Z 941.916,A -85,B 0,C 180,E1 22012.998,E2 22012.998} C_VEL
LIN {X 0,Y 473.321,Z 919.975,A -85,B 0,C 180,E1 22012.443,E2 22012.443} C_VEL
LIN {X 0,Y 478.123,Z 722.426,A -85,B 0,C 180,E1 22009.07,E2 22009.07} C_VEL
LIN {X 0,Y 465.522,Z 703.13,A -85,B 0,C 180,E1 22007.247,E2 22007.247} C_VEL
LIN {X 0,Y 458.115,Z 692.657,A -85,B 0,C 180,E1 22006.12,E2 22006.12} C_VEL
LIN {X 0,Y 455.451,Z 688.847,A -85,B 0,C 180,E1 22005.699,E2 22005.699} C_VEL
LIN {X 0,Y 452.829,Z 684.849,A -85,B 0,C 180,E1 22005.27,E2 22005.27} C_VEL
LIN {X 0,Y 449.926,Z 681.392,A -85,B 0,C 180,E1 22004.809,E2 22004.809} C_VEL
LIN {X 0,Y 449.225,Z 679.363,A -85,B 0,C 180,E1 22004.585,E2 22004.585} C_VEL
LIN {X 0,Y 449.131,Z 678.818,A -85,B 0,C 180,E1 22004.349,E2 22004.349} C_VEL
LIN {X 0,Y 449.132,Z 678.772,A -85,B 0,C 180,E1 22000.614,E2 22000.614} C_VEL
LIN {X 0,Y 449.123,Z 678.737,A -85,B 0,C 180,E1 21996.946,E2 21996.946} C_VEL
LIN {X 0,Y 449.13,Z 678.788,A -85,B 0,C 180,E1 21993.172,E2 21993.172} C_VEL
LIN {X 0,Y 449.127,Z 678.733,A -85,B 0,C 180,E1 21989.326,E2 21989.326} C_VEL
LIN {X 0,Y 449.128,Z 678.784,A -85,B 0,C 180,E1 21985.588,E2 21985.588} C_VEL
LIN {X 0,Y 449.13,Z 678.785,A -85,B 0,C 180,E1 21981.826,E2 21981.826} C_VEL
LIN {X 0,Y 449.138,Z 678.79,A -85,B 0,C 180,E1 21978.026,E2 21978.026} C_VEL
LIN {X 0,Y 449.14,Z 678.784,A -85,B 0,C 180,E1 21974.306,E2 21974.306} C_VEL
LIN {X 0,Y 449.126,Z 678.779,A -85,B 0,C 180,E1 21970.519,E2 21970.519} C_VEL
LIN {X 0,Y 449.129,Z 678.77,A -85,B 0,C 180,E1 21966.776,E2 21966.776} C_VEL
LIN {X 0,Y 449.13,Z 678.777,A -85,B 0,C 180,E1 21963.063,E2 21963.063} C_VEL
LIN {X 0,Y 449.142,Z 678.79,A -85,B 0,C 180,E1 21959.362,E2 21959.362} C_VEL
LIN {X 0,Y 449.124,Z 678.786,A -85,B 0,C 180,E1 21955.531,E2 21955.531} C_VEL
LIN {X 0,Y 449.132,Z 678.778,A -85,B 0,C 180,E1 21951.809,E2 21951.809} C_VEL
LIN {X 0,Y 449.122,Z 678.763,A -85,B 0,C 180,E1 21948.051,E2 21948.051} C_VEL
LIN {X 0,Y 449.135,Z 678.788,A -85,B 0,C 180,E1 21944.241,E2 21944.241} C_VEL
LIN {X 0,Y 449.121,Z 678.756,A -85,B 0,C 180,E1 21940.492,E2 21940.492} C_VEL
LIN {X 0,Y 449.134,Z 678.777,A -85,B 0,C 180,E1 21936.794,E2 21936.794} C_VEL
LIN {X 0,Y 449.125,Z 678.791,A -85,B 0,C 180,E1 21932.99,E2 21932.99} C_VEL
LIN {X 0,Y 449.135,Z 678.773,A -85,B 0,C 180,E1 21929.202,E2 21929.202} C_VEL
LIN {X 0,Y 449.124,Z 678.768,A -85,B 0,C 180,E1 21925.411,E2 21925.411} C_VEL
LIN {X 0,Y 449.161,Z 679.042,A -85,B 0,C 180,E1 21922.133,E2 21922.133} C_VEL
LIN {X 0,Y 450.486,Z 682.326,A -85,B 0,C 180,E1 21921.577,E2 21921.577} C_VEL
LIN {X 0,Y 455.926,Z 693.019,A -85,B 0,C 180,E1 21919.853,E2 21919.853} C_VEL
LIN {X 0,Y 463.444,Z 708.884,A -85,B 0,C 180,E1 21917.524,E2 21917.524} C_VEL
LIN {X 0,Y 471.858,Z 728.484,A -85,B 0,C 180,E1 21914.949,E2 21914.949} C_VEL
LIN {X 0,Y 473.234,Z 731.96,A -85,B 0,C 180,E1 21914.523,E2 21914.523} C_VEL
LIN {X 0,Y 472.37,Z 745.524,A -85,B 0,C 180,E1 21913.54,E2 21913.54} C_VEL
LIN {X 0,Y 478.368,Z 789.086,A -85,B 0,C 180,E1 21912.033,E2 21912.033} C_VEL
LIN {X 0,Y 473.178,Z 1018.787,A -85,B 0,C 180,E1 21908.174,E2 21908.174} C_VEL
LIN {X 0,Y 472.091,Z 1059.122,A -85,B 0,C 180,E1 21907.466,E2 21907.466} C_VEL
LIN {X 0,Y 470.654,Z 1081.273,A -85,B 0,C 180,E1 21906.884,E2 21906.884} C_VEL
LIN {X 0,Y 468.974,Z 1102.2,A -85,B 0,C 180,E1 21906.12,E2 21906.12} C_VEL
LIN {X 0,Y 467.056,Z 1122.931,A -85,B 0,C 180,E1 21905.159,E2 21905.159} C_VEL
LIN {X 0,Y 464.807,Z 1143.986,A -85,B 0,C 180,E1 21903.931,E2 21903.931} C_VEL
LIN {X 0,Y 462.496,Z 1164.266,A -85,B 0,C 180,E1 21902.501,E2 21902.501} C_VEL
LIN {X 0,Y 460.201,Z 1183.655,A -85,B 0,C 180,E1 21900.886,E2 21900.886} C_VEL
LIN {X 0,Y 457.958,Z 1202.284,A -85,B 0,C 180,E1 21899.053,E2 21899.053} C_VEL
LIN {X 0,Y 455.859,Z 1219.632,A -85,B 0,C 180,E1 21897.064,E2 21897.064} C_VEL
LIN {X 0,Y 453.926,Z 1236.142,A -85,B 0,C 180,E1 21894.879,E2 21894.879} C_VEL
LIN {X 0,Y 452.305,Z 1250.846,A -85,B 0,C 180,E1 21892.621,E2 21892.621} C_VEL
LIN {X 0,Y 451.013,Z 1263.43,A -85,B 0,C 180,E1 21890.368,E2 21890.368} C_VEL
LIN {X 0,Y 450.018,Z 1273.102,A -85,B 0,C 180,E1 21888.256,E2 21888.256} C_VEL
LIN {X 0,Y 449.099,Z 1283.133,A -85,B 0,C 180,E1 21885.627,E2 21885.627} C_VEL
LIN {X 0,Y 448.494,Z 1291.762,A -85,B 0,C 180,E1 21882.881,E2 21882.881} C_VEL
LIN {X 0,Y 448.164,Z 1298.28,A -85,B 0,C 180,E1 21880.281,E2 21880.281} C_VEL
LIN {X 0,Y 447.987,Z 1303.399,A -85,B 0,C 180,E1 21877.567,E2 21877.567} C_VEL
LIN {X 0,Y 447.918,Z 1306.99,A -85,B 0,C 180,E1 21874.866,E2 21874.866} C_VEL
LIN {X 0,Y 447.906,Z 1308.881,A -85,B 0,C 180,E1 21872.303,E2 21872.303} C_VEL
LIN {X 0,Y 447.896,Z 1309.416,A -85,B 0,C 180,E1 21869.488,E2 21869.488} C_VEL
LIN {X 0,Y 447.907,Z 1308.471,A -85,B 0,C 180,E1 21866.929,E2 21866.929} C_VEL
LIN {X 0,Y 447.933,Z 1305.935,A -85,B 0,C 180,E1 21864.235,E2 21864.235} C_VEL
LIN {X 0,Y 448.021,Z 1301.923,A -85,B 0,C 180,E1 21861.53,E2 21861.53} C_VEL
LIN {X 0,Y 448.232,Z 1296.462,A -85,B 0,C 180,E1 21858.94,E2 21858.94} C_VEL
LIN {X 0,Y 448.695,Z 1288.69,A -85,B 0,C 180,E1 21856.075,E2 21856.075} C_VEL
LIN {X 0,Y 449.391,Z 1279.893,A -85,B 0,C 180,E1 21853.454,E2 21853.454} C_VEL
LIN {X 0,Y 450.429,Z 1269.09,A -85,B 0,C 180,E1 21850.821,E2 21850.821} C_VEL
LIN {X 0,Y 451.502,Z 1258.513,A -85,B 0,C 180,E1 21848.705,E2 21848.705} C_VEL
LIN {X 0,Y 453.039,Z 1244.221,A -85,B 0,C 180,E1 21846.318,E2 21846.318} C_VEL
LIN {X 0,Y 454.827,Z 1228.408,A -85,B 0,C 180,E1 21844.058,E2 21844.058} C_VEL
LIN {X 0,Y 456.948,Z 1210.568,A -85,B 0,C 180,E1 21841.861,E2 21841.861} C_VEL
LIN {X 0,Y 459.139,Z 1192.471,A -85,B 0,C 180,E1 21839.944,E2 21839.944} C_VEL
LIN {X 0,Y 461.434,Z 1173.429,A -85,B 0,C 180,E1 21838.229,E2 21838.229} C_VEL
LIN {X 0,Y 463.705,Z 1153.673,A -85,B 0,C 180,E1 21836.719,E2 21836.719} C_VEL
LIN {X 0,Y 466.012,Z 1133.011,A -85,B 0,C 180,E1 21835.398,E2 21835.398} C_VEL
LIN {X 0,Y 468.042,Z 1112.432,A -85,B 0,C 180,E1 21834.325,E2 21834.325} C_VEL
LIN {X 0,Y 469.933,Z 1090.819,A -85,B 0,C 180,E1 21833.44,E2 21833.44} C_VEL
LIN {X 0,Y 471.516,Z 1069.169,A -85,B 0,C 180,E1 21832.772,E2 21832.772} C_VEL
LIN {X 0,Y 472.561,Z 1046.656,A -85,B 0,C 180,E1 21832.293,E2 21832.293} C_VEL
LIN {X 0,Y 477.532,Z 823.879,A -85,B 0,C 180,E1 21828.556,E2 21828.556} C_VEL
LIN {X 0,Y 478.229,Z 786.784,A -85,B 0,C 180,E1 21827.909,E2 21827.909} C_VEL
LIN {X 0,Y 472.296,Z 744.788,A -85,B 0,C 180,E1 21826.431,E2 21826.431} C_VEL
LIN {X 0,Y 473.11,Z 731.672,A -85,B 0,C 180,E1 21825.443,E2 21825.443} C_VEL
LIN {X 0,Y 465.033,Z 712.41,A -85,B 0,C 180,E1 21822.967,E2 21822.967} C_VEL
LIN {X 0,Y 457.108,Z 695.336,A -85,B 0,C 180,E1 21820.515,E2 21820.515} C_VEL
LIN {X 0,Y 450.9,Z 682.912,A -85,B 0,C 180,E1 21818.543,E2 21818.543} C_VEL
LIN {X 0,Y 449.183,Z 679.169,A -85,B 0,C 180,E1 21817.905,E2 21817.905} C_VEL
LIN {X 0,Y 449.128,Z 678.771,A -85,B 0,C 180,E1 21816.947,E2 21816.947} C_VEL
LIN {X 0,Y 449.125,Z 678.769,A -85,B 0,C 180,E1 21813.171,E2 21813.171} C_VEL
LIN {X 0,Y 449.13,Z 678.76,A -85,B 0,C 180,E1 21809.471,E2 21809.471} C_VEL
LIN {X 0,Y 449.123,Z 678.771,A -85,B 0,C 180,E1 21805.729,E2 21805.729} C_VEL
LIN {X 0,Y 449.134,Z 678.791,A -85,B 0,C 180,E1 21801.962,E2 21801.962} C_VEL
LIN {X 0,Y 449.124,Z 678.763,A -85,B 0,C 180,E1 21798.16,E2 21798.16} C_VEL
LIN {X 0,Y 449.132,Z 678.769,A -85,B 0,C 180,E1 21794.438,E2 21794.438} C_VEL
LIN {X 0,Y 449.124,Z 678.787,A -85,B 0,C 180,E1 21790.648,E2 21790.648} C_VEL
LIN {X 0,Y 449.133,Z 678.776,A -85,B 0,C 180,E1 21786.854,E2 21786.854} C_VEL
LIN {X 0,Y 449.127,Z 678.775,A -85,B 0,C 180,E1 21783.19,E2 21783.19} C_VEL
LIN {X 0,Y 449.134,Z 678.785,A -85,B 0,C 180,E1 21779.362,E2 21779.362} C_VEL
LIN {X 0,Y 449.123,Z 678.788,A -85,B 0,C 180,E1 21775.659,E2 21775.659} C_VEL
LIN {X 0,Y 449.139,Z 678.784,A -85,B 0,C 180,E1 21771.938,E2 21771.938} C_VEL
LIN {X 0,Y 449.134,Z 678.774,A -85,B 0,C 180,E1 21768.181,E2 21768.181} C_VEL
LIN {X 0,Y 449.131,Z 678.776,A -85,B 0,C 180,E1 21764.505,E2 21764.505} C_VEL
LIN {X 0,Y 449.125,Z 678.783,A -85,B 0,C 180,E1 21760.716,E2 21760.716} C_VEL
LIN {X 0,Y 449.139,Z 678.782,A -85,B 0,C 180,E1 21756.933,E2 21756.933} C_VEL
LIN {X 0,Y 449.135,Z 678.785,A -85,B 0,C 180,E1 21753.133,E2 21753.133} C_VEL
LIN {X 0,Y 449.124,Z 678.729,A -85,B 0,C 180,E1 21749.489,E2 21749.489} C_VEL
LIN {X 0,Y 449.126,Z 678.786,A -85,B 0,C 180,E1 21745.68,E2 21745.68} C_VEL
LIN {X 0,Y 449.127,Z 678.747,A -85,B 0,C 180,E1 21741.927,E2 21741.927} C_VEL
LIN {X 0,Y 449.123,Z 678.747,A -85,B 0,C 180,E1 21738.225,E2 21738.225} C_VEL
LIN {X 0,Y 449.157,Z 678.976,A -85,B 0,C 180,E1 21735.424,E2 21735.424} C_VEL
LIN {X 0,Y 449.518,Z 680.431,A -85,B 0,C 180,E1 21735.178,E2 21735.178} C_VEL
LIN {X 0,Y 451.528,Z 683.577,A -85,B 0,C 180,E1 21734.833,E2 21734.833} C_VEL
LIN {X 0,Y 452.956,Z 685.143,A -85,B 0,C 180,E1 21734.611,E2 21734.611} C_VEL
LIN {X 0,Y 455.595,Z 689.001,A -85,B 0,C 180,E1 21734.185,E2 21734.185} C_VEL
LIN {X 0,Y 466.476,Z 704.553,A -85,B 0,C 180,E1 21732.517,E2 21732.517} C_VEL
LIN {X 0,Y 478.186,Z 722.542,A -85,B 0,C 180,E1 21730.829,E2 21730.829} C_VEL
LIN {X 0,Y 473.902,Z 897.452,A -85,B 0,C 180,E1 21727.866,E2 21727.866} C_VEL
LIN {X 0,Y 472.905,Z 905.153,A -85,B 0,C 180,E1 21727.818,E2 21727.818} C_VEL
LIN {X 0,Y 467.45,Z 925.658,A -85,B 0,C 180,E1 21727.92,E2 21727.92} C_VEL
LIN {X 0,Y 466.681,Z 931.104,A -85,B 0,C 180,E1 21727.839,E2 21727.839} C_VEL
LIN {X 0,Y 466.625,Z 932.19,A -85,B 0,C 180,E1 21727.811,E2 21727.811} C_VEL
LIN {X 0,Y 465.469,Z 953.539,A -85,B 0,C 180,E1 21727.156,E2 21727.156} C_VEL
LIN {X 0,Y 463.931,Z 973.023,A -85,B 0,C 180,E1 21726.346,E2 21726.346} C_VEL
LIN {X 0,Y 461.833,Z 993.998,A -85,B 0,C 180,E1 21725.236,E2 21725.236} C_VEL
LIN {X 0,Y 459.609,Z 1013.008,A -85,B 0,C 180,E1 21723.992,E2 21723.992} C_VEL
LIN {X 0,Y 457.157,Z 1031.115,A -85,B 0,C 180,E1 21722.549,E2 21722.549} C_VEL
LIN {X 0,Y 454.445,Z 1049.1,A -85,B 0,C 180,E1 21720.839,E2 21720.839} C_VEL
LIN {X 0,Y 451.852,Z 1065.548,A -85,B 0,C 180,E1 21718.986,E2 21718.986} C_VEL
LIN {X 0,Y 449.287,Z 1081.019,A -85,B 0,C 180,E1 21716.927,E2 21716.927} C_VEL
LIN {X 0,Y 446.955,Z 1094.969,A -85,B 0,C 180,E1 21714.728,E2 21714.728} C_VEL
LIN {X 0,Y 444.76,Z 1108.597,A -85,B 0,C 180,E1 21712.189,E2 21712.189} C_VEL
LIN {X 0,Y 443.047,Z 1120.052,A -85,B 0,C 180,E1 21709.649,E2 21709.649} C_VEL
LIN {X 0,Y 441.701,Z 1130.027,A -85,B 0,C 180,E1 21706.978,E2 21706.978} C_VEL
LIN {X 0,Y 440.641,Z 1140.576,A -85,B 0,C 180,E1 21703.516,E2 21703.516} C_VEL
LIN {X 0,Y 440.217,Z 1147.573,A -85,B 0,C 180,E1 21700.733,E2 21700.733} C_VEL
LIN {X 0,Y 440.007,Z 1153.122,A -85,B 0,C 180,E1 21697.836,E2 21697.836} C_VEL
LIN {X 0,Y 439.916,Z 1156.833,A -85,B 0,C 180,E1 21695.085,E2 21695.085} C_VEL
LIN {X 0,Y 439.902,Z 1158.858,A -85,B 0,C 180,E1 21692.345,E2 21692.345} C_VEL
LIN {X 0,Y 439.898,Z 1159.423,A -85,B 0,C 180,E1 21689.479,E2 21689.479} C_VEL
LIN {X 0,Y 439.907,Z 1158.497,A -85,B 0,C 180,E1 21686.873,E2 21686.873} C_VEL
LIN {X 0,Y 439.938,Z 1155.995,A -85,B 0,C 180,E1 21684.13,E2 21684.13} C_VEL
LIN {X 0,Y 440.041,Z 1152.01,A -85,B 0,C 180,E1 21681.375,E2 21681.375} C_VEL
LIN {X 0,Y 440.287,Z 1146.26,A -85,B 0,C 180,E1 21678.605,E2 21678.605} C_VEL
LIN {X 0,Y 440.787,Z 1138.443,A -85,B 0,C 180,E1 21675.686,E2 21675.686} C_VEL
LIN {X 0,Y 441.773,Z 1129.401,A -85,B 0,C 180,E1 21672.754,E2 21672.754} C_VEL
LIN {X 0,Y 443.156,Z 1119.339,A -85,B 0,C 180,E1 21670.082,E2 21670.082} C_VEL
LIN {X 0,Y 444.902,Z 1107.718,A -85,B 0,C 180,E1 21667.54,E2 21667.54} C_VEL
LIN {X 0,Y 447.002,Z 1094.689,A -85,B 0,C 180,E1 21665.133,E2 21665.133} C_VEL
LIN {X 0,Y 449.343,Z 1080.674,A -85,B 0,C 180,E1 21662.933,E2 21662.933} C_VEL
LIN {X 0,Y 451.837,Z 1065.654,A -85,B 0,C 180,E1 21660.937,E2 21660.937} C_VEL
LIN {X 0,Y 454.38,Z 1049.525,A -85,B 0,C 180,E1 21659.114,E2 21659.114} C_VEL
LIN {X 0,Y 457.033,Z 1032.058,A -85,B 0,C 180,E1 21657.441,E2 21657.441} C_VEL
LIN {X 0,Y 459.466,Z 1014.047,A -85,B 0,C 180,E1 21655.996,E2 21655.996} C_VEL
LIN {X 0,Y 461.745,Z 994.803,A -85,B 0,C 180,E1 21654.722,E2 21654.722} C_VEL
LIN {X 0,Y 463.795,Z 974.713,A -85,B 0,C 180,E1 21653.642,E2 21653.642} C_VEL
LIN {X 0,Y 465.329,Z 955.399,A -85,B 0,C 180,E1 21652.826,E2 21652.826} C_VEL
LIN {X 0,Y 466.568,Z 933.529,A -85,B 0,C 180,E1 21652.134,E2 21652.134} C_VEL
LIN {X 0,Y 467.387,Z 910.506,A -85,B 0,C 180,E1 21651.645,E2 21651.645} C_VEL
LIN {X 0,Y 472.11,Z 725.782,A -85,B 0,C 180,E1 21648.475,E2 21648.475} C_VEL
LIN {X 0,Y 458.164,Z 704.59,A -85,B 0,C 180,E1 21646.385,E2 21646.385} C_VEL
LIN {X 0,Y 450.793,Z 694.329,A -85,B 0,C 180,E1 21645.216,E2 21645.216} C_VEL
LIN {X 0,Y 447.71,Z 690.014,A -85,B 0,C 180,E1 21644.707,E2 21644.707} C_VEL
LIN {X 0,Y 445.058,Z 686.057,A -85,B 0,C 180,E1 21644.255,E2 21644.255} C_VEL
LIN {X 0,Y 441.988,Z 682.36,A -85,B 0,C 180,E1 21643.74,E2 21643.74} C_VEL
LIN {X 0,Y 441.316,Z 680.468,A -85,B 0,C 180,E1 21643.532,E2 21643.532} C_VEL
LIN {X 0,Y 441.191,Z 679.774,A -85,B 0,C 180,E1 21643.19,E2 21643.19} C_VEL
LIN {X 0,Y 441.198,Z 679.774,A -85,B 0,C 180,E1 21639.387,E2 21639.387} C_VEL
LIN {X 0,Y 441.181,Z 679.738,A -85,B 0,C 180,E1 21635.552,E2 21635.552} C_VEL
LIN {X 0,Y 441.19,Z 679.738,A -85,B 0,C 180,E1 21631.807,E2 21631.807} C_VEL
LIN {X 0,Y 441.183,Z 679.75,A -85,B 0,C 180,E1 21627.978,E2 21627.978} C_VEL
LIN {X 0,Y 441.196,Z 679.762,A -85,B 0,C 180,E1 21624.217,E2 21624.217} C_VEL
LIN {X 0,Y 441.198,Z 679.761,A -85,B 0,C 180,E1 21620.426,E2 21620.426} C_VEL
LIN {X 0,Y 441.198,Z 679.765,A -85,B 0,C 180,E1 21616.592,E2 21616.592} C_VEL
LIN {X 0,Y 441.185,Z 679.775,A -85,B 0,C 180,E1 21612.832,E2 21612.832} C_VEL
LIN {X 0,Y 441.192,Z 679.777,A -85,B 0,C 180,E1 21608.997,E2 21608.997} C_VEL
LIN {X 0,Y 441.193,Z 679.773,A -85,B 0,C 180,E1 21605.201,E2 21605.201} C_VEL
LIN {X 0,Y 441.199,Z 679.759,A -85,B 0,C 180,E1 21601.429,E2 21601.429} C_VEL
LIN {X 0,Y 441.186,Z 679.763,A -85,B 0,C 180,E1 21597.662,E2 21597.662} C_VEL
LIN {X 0,Y 441.19,Z 679.772,A -85,B 0,C 180,E1 21593.886,E2 21593.886} C_VEL
LIN {X 0,Y 441.189,Z 679.778,A -85,B 0,C 180,E1 21590.082,E2 21590.082} C_VEL
LIN {X 0,Y 441.187,Z 679.745,A -85,B 0,C 180,E1 21586.234,E2 21586.234} C_VEL
LIN {X 0,Y 441.186,Z 679.765,A -85,B 0,C 180,E1 21582.57,E2 21582.57} C_VEL
LIN {X 0,Y 441.19,Z 679.775,A -85,B 0,C 180,E1 21578.74,E2 21578.74} C_VEL
LIN {X 0,Y 441.185,Z 679.749,A -85,B 0,C 180,E1 21575.025,E2 21575.025} C_VEL
LIN {X 0,Y 441.193,Z 679.754,A -85,B 0,C 180,E1 21571.284,E2 21571.284} C_VEL
LIN {X 0,Y 441.186,Z 679.769,A -85,B 0,C 180,E1 21567.513,E2 21567.513} C_VEL
LIN {X 0,Y 441.19,Z 679.772,A -85,B 0,C 180,E1 21563.737,E2 21563.737} C_VEL
LIN {X 0,Y 441.261,Z 680.229,A -85,B 0,C 180,E1 21563.102,E2 21563.102} C_VEL
LIN {X 0,Y 442.552,Z 683.326,A -85,B 0,C 180,E1 21562.573,E2 21562.573} C_VEL
LIN {X 0,Y 443.721,Z 685.394,A -85,B 0,C 180,E1 21562.2,E2 21562.2} C_VEL
LIN {X 0,Y 450.587,Z 699.182,A -85,B 0,C 180,E1 21559.946,E2 21559.946} C_VEL
LIN {X 0,Y 458.446,Z 715.993,A -85,B 0,C 180,E1 21557.461,E2 21557.461} C_VEL
LIN {X 0,Y 466.457,Z 735.218,A -85,B 0,C 180,E1 21554.932,E2 21554.932} C_VEL
LIN {X 0,Y 465.996,Z 744.009,A -85,B 0,C 180,E1 21554.289,E2 21554.289} C_VEL
LIN {X 0,Y 472.29,Z 790.436,A -85,B 0,C 180,E1 21552.646,E2 21552.646} C_VEL
LIN {X 0,Y 466.768,Z 1019.986,A -85,B 0,C 180,E1 21548.745,E2 21548.745} C_VEL
LIN {X 0,Y 465.66,Z 1058.025,A -85,B 0,C 180,E1 21548.065,E2 21548.065} C_VEL
LIN {X 0,Y 464.137,Z 1080.101,A -85,B 0,C 180,E1 21547.48,E2 21547.48} C_VEL
LIN {X 0,Y 462.291,Z 1101.466,A -85,B 0,C 180,E1 21546.69,E2 21546.69} C_VEL
LIN {X 0,Y 460.184,Z 1122.637,A -85,B 0,C 180,E1 21545.687,E2 21545.687} C_VEL
LIN {X 0,Y 457.916,Z 1142.515,A -85,B 0,C 180,E1 21544.513,E2 21544.513} C_VEL
LIN {X 0,Y 455.433,Z 1162.87,A -85,B 0,C 180,E1 21543.062,E2 21543.062} C_VEL
LIN {X 0,Y 452.944,Z 1182.552,A -85,B 0,C 180,E1 21541.396,E2 21541.396} C_VEL
LIN {X 0,Y 450.529,Z 1201.349,A -85,B 0,C 180,E1 21539.516,E2 21539.516} C_VEL
LIN {X 0,Y 448.276,Z 1218.621,A -85,B 0,C 180,E1 21537.496,E2 21537.496} C_VEL
LIN {X 0,Y 446.173,Z 1235.559,A -85,B 0,C 180,E1 21535.199,E2 21535.199} C_VEL
LIN {X 0,Y 444.475,Z 1250.191,A -85,B 0,C 180,E1 21532.902,E2 21532.902} C_VEL
LIN {X 0,Y 443.052,Z 1263.386,A -85,B 0,C 180,E1 21530.474,E2 21530.474} C_VEL
LIN {X 0,Y 441.845,Z 1275.881,A -85,B 0,C 180,E1 21527.787,E2 21527.787} C_VEL
LIN {X 0,Y 441.212,Z 1283.122,A -85,B 0,C 180,E1 21525.914,E2 21525.914} C_VEL
LIN {X 0,Y 440.563,Z 1291.564,A -85,B 0,C 180,E1 21523.192,E2 21523.192} C_VEL
LIN {X 0,Y 440.198,Z 1297.977,A -85,B 0,C 180,E1 21520.601,E2 21520.601} C_VEL
LIN {X 0,Y 440.007,Z 1303.249,A -85,B 0,C 180,E1 21517.8,E2 21517.8} C_VEL
LIN {X 0,Y 439.922,Z 1306.876,A -85,B 0,C 180,E1 21515.085,E2 21515.085} C_VEL
LIN {X 0,Y 439.905,Z 1308.881,A -85,B 0,C 180,E1 21512.345,E2 21512.345} C_VEL
LIN {X 0,Y 439.896,Z 1309.416,A -85,B 0,C 180,E1 21509.479,E2 21509.479} C_VEL
LIN {X 0,Y 439.909,Z 1308.47,A -85,B 0,C 180,E1 21506.873,E2 21506.873} C_VEL
LIN {X 0,Y 439.933,Z 1305.935,A -85,B 0,C 180,E1 21504.13,E2 21504.13} C_VEL
LIN {X 0,Y 440.036,Z 1301.923,A -85,B 0,C 180,E1 21501.375,E2 21501.375} C_VEL
LIN {X 0,Y 440.269,Z 1296.462,A -85,B 0,C 180,E1 21498.738,E2 21498.738} C_VEL
LIN {X 0,Y 440.77,Z 1288.69,A -85,B 0,C 180,E1 21495.819,E2 21495.819} C_VEL
LIN {X 0,Y 441.432,Z 1280.754,A -85,B 0,C 180,E1 21493.418,E2 21493.418} C_VEL
LIN {X 0,Y 442.335,Z 1270.526,A -85,B 0,C 180,E1 21491.005,E2 21491.005} C_VEL
LIN {X 0,Y 443.555,Z 1258.546,A -85,B 0,C 180,E1 21488.582,E2 21488.582} C_VEL
LIN {X 0,Y 445.196,Z 1243.909,A -85,B 0,C 180,E1 21486.074,E2 21486.074} C_VEL
LIN {X 0,Y 447.119,Z 1227.906,A -85,B 0,C 180,E1 21483.72,E2 21483.72} C_VEL
LIN {X 0,Y 449.331,Z 1210.502,A -85,B 0,C 180,E1 21481.517,E2 21481.517} C_VEL
LIN {X 0,Y 451.692,Z 1192.359,A -85,B 0,C 180,E1 21479.543,E2 21479.543} C_VEL
LIN {X 0,Y 454.105,Z 1173.484,A -85,B 0,C 180,E1 21477.804,E2 21477.804} C_VEL
LIN {X 0,Y 456.635,Z 1153.135,A -85,B 0,C 180,E1 21476.21,E2 21476.21} C_VEL
LIN {X 0,Y 459.036,Z 1133.13,A -85,B 0,C 180,E1 21474.899,E2 21474.899} C_VEL
LIN {X 0,Y 461.304,Z 1111.638,A -85,B 0,C 180,E1 21473.761,E2 21473.761} C_VEL
LIN {X 0,Y 463.355,Z 1089.821,A -85,B 0,C 180,E1 21472.854,E2 21472.854} C_VEL
LIN {X 0,Y 465.024,Z 1068.553,A -85,B 0,C 180,E1 21472.186,E2 21472.186} C_VEL
LIN {X 0,Y 466.144,Z 1045.9,A -85,B 0,C 180,E1 21471.696,E2 21471.696} C_VEL
LIN {X 0,Y 471.434,Z 823.872,A -85,B 0,C 180,E1 21467.927,E2 21467.927} C_VEL
LIN {X 0,Y 472.155,Z 788.259,A -85,B 0,C 180,E1 21467.298,E2 21467.298} C_VEL
LIN {X 0,Y 465.934,Z 742.821,A -85,B 0,C 180,E1 21465.652,E2 21465.652} C_VEL
LIN {X 0,Y 466.341,Z 734.931,A -85,B 0,C 180,E1 21465.034,E2 21465.034} C_VEL
LIN {X 0,Y 458.26,Z 715.571,A -85,B 0,C 180,E1 21462.486,E2 21462.486} C_VEL
LIN {X 0,Y 449.652,Z 697.041,A -85,B 0,C 180,E1 21459.739,E2 21459.739} C_VEL
LIN {X 0,Y 442.956,Z 683.883,A -85,B 0,C 180,E1 21457.55,E2 21457.55} C_VEL
LIN {X 0,Y 441.244,Z 680.136,A -85,B 0,C 180,E1 21456.882,E2 21456.882} C_VEL
LIN {X 0,Y 441.184,Z 679.777,A -85,B 0,C 180,E1 21455.622,E2 21455.622} C_VEL
LIN {X 0,Y 441.196,Z 679.78,A -85,B 0,C 180,E1 21451.808,E2 21451.808} C_VEL
LIN {X 0,Y 441.185,Z 679.769,A -85,B 0,C 180,E1 21447.977,E2 21447.977} C_VEL
LIN {X 0,Y 441.19,Z 679.749,A -85,B 0,C 180,E1 21444.217,E2 21444.217} C_VEL
LIN {X 0,Y 441.185,Z 679.76,A -85,B 0,C 180,E1 21440.565,E2 21440.565} C_VEL
LIN {X 0,Y 441.192,Z 679.775,A -85,B 0,C 180,E1 21436.727,E2 21436.727} C_VEL
LIN {X 0,Y 441.181,Z 679.741,A -85,B 0,C 180,E1 21432.965,E2 21432.965} C_VEL
LIN {X 0,Y 441.195,Z 679.774,A -85,B 0,C 180,E1 21429.128,E2 21429.128} C_VEL
LIN {X 0,Y 441.188,Z 679.777,A -85,B 0,C 180,E1 21425.462,E2 21425.462} C_VEL
LIN {X 0,Y 441.192,Z 679.768,A -85,B 0,C 180,E1 21421.688,E2 21421.688} C_VEL
LIN {X 0,Y 441.183,Z 679.759,A -85,B 0,C 180,E1 21417.922,E2 21417.922} C_VEL
LIN {X 0,Y 441.198,Z 679.762,A -85,B 0,C 180,E1 21414.147,E2 21414.147} C_VEL
LIN {X 0,Y 441.197,Z 679.775,A -85,B 0,C 180,E1 21410.327,E2 21410.327} C_VEL
LIN {X 0,Y 441.196,Z 679.777,A -85,B 0,C 180,E1 21406.456,E2 21406.456} C_VEL
LIN {X 0,Y 441.185,Z 679.772,A -85,B 0,C 180,E1 21402.729,E2 21402.729} C_VEL
LIN {X 0,Y 441.199,Z 679.764,A -85,B 0,C 180,E1 21399.012,E2 21399.012} C_VEL
LIN {X 0,Y 441.196,Z 679.763,A -85,B 0,C 180,E1 21395.212,E2 21395.212} C_VEL
LIN {X 0,Y 441.196,Z 679.735,A -85,B 0,C 180,E1 21391.433,E2 21391.433} C_VEL
LIN {X 0,Y 441.183,Z 679.753,A -85,B 0,C 180,E1 21387.666,E2 21387.666} C_VEL
LIN {X 0,Y 441.189,Z 679.728,A -85,B 0,C 180,E1 21383.897,E2 21383.897} C_VEL
LIN {X 0,Y 441.188,Z 679.781,A -85,B 0,C 180,E1 21380.106,E2 21380.106} C_VEL
LIN {X 0,Y 441.216,Z 679.942,A -85,B 0,C 180,E1 21376.507,E2 21376.507} C_VEL
LIN {X 0,Y 441.574,Z 681.387,A -85,B 0,C 180,E1 21376.251,E2 21376.251} C_VEL
LIN {X 0,Y 443.549,Z 684.497,A -85,B 0,C 180,E1 21375.894,E2 21375.894} C_VEL
LIN {X 0,Y 445.035,Z 686.016,A -85,B 0,C 180,E1 21375.653,E2 21375.653} C_VEL
LIN {X 0,Y 447.688,Z 689.996,A -85,B 0,C 180,E1 21375.2,E2 21375.2} C_VEL
LIN {X 0,Y 449.842,Z 693.046,A -85,B 0,C 180,E1 21374.843,E2 21374.843} C_VEL
LIN {X 0,Y 456.096,Z 701.689,A -85,B 0,C 180,E1 21373.843,E2 21373.843} C_VEL
LIN {X 0,Y 468.86,Z 720.735,A -85,B 0,C 180,E1 21371.905,E2 21371.905} C_VEL
LIN {X 0,Y 472.173,Z 726.256,A -85,B 0,C 180,E1 21371.417,E2 21371.417} C_VEL
LIN {X 0,Y 466.969,Z 924.903,A -85,B 0,C 180,E1 21367.986,E2 21367.986} C_VEL
LIN {X 0,Y 466.625,Z 932.19,A -85,B 0,C 180,E1 21367.811,E2 21367.811} C_VEL
LIN {X 0,Y 465.476,Z 939.811,A -85,B 0,C 180,E1 21367.693,E2 21367.693} C_VEL
LIN {X 0,Y 459.681,Z 959.019,A -85,B 0,C 180,E1 21367.521,E2 21367.521} C_VEL
LIN {X 0,Y 458.319,Z 966.422,A -85,B 0,C 180,E1 21367.299,E2 21367.299} C_VEL
LIN {X 0,Y 456.45,Z 986.155,A -85,B 0,C 180,E1 21366.336,E2 21366.336} C_VEL
LIN {X 0,Y 454.197,Z 1005.822,A -85,B 0,C 180,E1 21365.145,E2 21365.145} C_VEL
LIN {X 0,Y 451.799,Z 1023.921,A -85,B 0,C 180,E1 21363.819,E2 21363.819} C_VEL
LIN {X 0,Y 449.044,Z 1042.067,A -85,B 0,C 180,E1 21362.207,E2 21362.207} C_VEL
LIN {X 0,Y 446.205,Z 1059.413,A -85,B 0,C 180,E1 21360.377,E2 21360.377} C_VEL
LIN {X 0,Y 443.494,Z 1075.271,A -85,B 0,C 180,E1 21358.404,E2 21358.404} C_VEL
LIN {X 0,Y 440.907,Z 1089.887,A -85,B 0,C 180,E1 21356.244,E2 21356.244} C_VEL
LIN {X 0,Y 438.514,Z 1103.407,A -85,B 0,C 180,E1 21353.89,E2 21353.89} C_VEL
LIN {X 0,Y 436.454,Z 1115.689,A -85,B 0,C 180,E1 21351.361,E2 21351.361} C_VEL
LIN {X 0,Y 434.849,Z 1126.197,A -85,B 0,C 180,E1 21348.778,E2 21348.778} C_VEL
LIN {X 0,Y 433.579,Z 1135.285,A -85,B 0,C 180,E1 21346.064,E2 21346.064} C_VEL
LIN {X 0,Y 432.692,Z 1143.355,A -85,B 0,C 180,E1 21343.088,E2 21343.088} C_VEL
LIN {X 0,Y 432.197,Z 1149.377,A -85,B 0,C 180,E1 21340.261,E2 21340.261} C_VEL
LIN {X 0,Y 431.97,Z 1154.925,A -85,B 0,C 180,E1 21336.779,E2 21336.779} C_VEL
LIN {X 0,Y 431.909,Z 1157.747,A -85,B 0,C 180,E1 21334.115,E2 21334.115} C_VEL
LIN {X 0,Y 431.906,Z 1159.294,A -85,B 0,C 180,E1 21331.194,E2 21331.194} C_VEL
LIN {X 0,Y 431.902,Z 1159.265,A -85,B 0,C 180,E1 21328.541,E2 21328.541} C_VEL
LIN {X 0,Y 431.914,Z 1157.711,A -85,B 0,C 180,E1 21325.752,E2 21325.752} C_VEL
LIN {X 0,Y 431.967,Z 1154.704,A -85,B 0,C 180,E1 21322.954,E2 21322.954} C_VEL
LIN {X 0,Y 432.224,Z 1149.048,A -85,B 0,C 180,E1 21319.467,E2 21319.467} C_VEL
LIN {X 0,Y 432.751,Z 1142.793,A -85,B 0,C 180,E1 21316.584,E2 21316.584} C_VEL
LIN {X 0,Y 433.601,Z 1135.143,A -85,B 0,C 180,E1 21313.799,E2 21313.799} C_VEL
LIN {X 0,Y 434.877,Z 1126.015,A -85,B 0,C 180,E1 21311.085,E2 21311.085} C_VEL
LIN {X 0,Y 436.557,Z 1115.11,A -85,B 0,C 180,E1 21308.415,E2 21308.415} C_VEL
LIN {X 0,Y 438.605,Z 1102.875,A -85,B 0,C 180,E1 21305.918,E2 21305.918} C_VEL
LIN {X 0,Y 441.112,Z 1088.698,A -85,B 0,C 180,E1 21303.479,E2 21303.479} C_VEL
LIN {X 0,Y 443.738,Z 1073.893,A -85,B 0,C 180,E1 21301.319,E2 21301.319} C_VEL
LIN {X 0,Y 446.451,Z 1058.02,A -85,B 0,C 180,E1 21299.37,E2 21299.37} C_VEL
LIN {X 0,Y 449.264,Z 1040.628,A -85,B 0,C 180,E1 21297.565,E2 21297.565} C_VEL
LIN {X 0,Y 452.005,Z 1022.347,A -85,B 0,C 180,E1 21295.97,E2 21295.97} C_VEL
LIN {X 0,Y 454.433,Z 1004.053,A -85,B 0,C 180,E1 21294.645,E2 21294.645} C_VEL
LIN {X 0,Y 456.625,Z 984.345,A -85,B 0,C 180,E1 21293.476,E2 21293.476} C_VEL
LIN {X 0,Y 458.528,Z 963.669,A -85,B 0,C 180,E1 21292.499,E2 21292.499} C_VEL
LIN {X 0,Y 459.959,Z 943.257,A -85,B 0,C 180,E1 21291.769,E2 21291.769} C_VEL
LIN {X 0,Y 460.894,Z 921.966,A -85,B 0,C 180,E1 21291.228,E2 21291.228} C_VEL
LIN {X 0,Y 466.156,Z 729.313,A -85,B 0,C 180,E1 21287.868,E2 21287.868} C_VEL
LIN {X 0,Y 453.467,Z 709.977,A -85,B 0,C 180,E1 21285.911,E2 21285.911} C_VEL
LIN {X 0,Y 443.579,Z 696.077,A -85,B 0,C 180,E1 21284.283,E2 21284.283} C_VEL
LIN {X 0,Y 439.945,Z 691.104,A -85,B 0,C 180,E1 21283.656,E2 21283.656} C_VEL
LIN {X 0,Y 437.272,Z 687.186,A -85,B 0,C 180,E1 21283.178,E2 21283.178} C_VEL
LIN {X 0,Y 434.045,Z 683.325,A -85,B 0,C 180,E1 21282.607,E2 21282.607} C_VEL
LIN {X 0,Y 433.345,Z 681.312,A -85,B 0,C 180,E1 21282.356,E2 21282.356} C_VEL
LIN {X 0,Y 433.246,Z 680.748,A -85,B 0,C 180,E1 21282.004,E2 21282.004} C_VEL
LIN {X 0,Y 433.252,Z 680.723,A -85,B 0,C 180,E1 21278.206,E2 21278.206} C_VEL
LIN {X 0,Y 433.246,Z 680.755,A -85,B 0,C 180,E1 21274.432,E2 21274.432} C_VEL
LIN {X 0,Y 433.25,Z 680.702,A -85,B 0,C 180,E1 21270.595,E2 21270.595} C_VEL
LIN {X 0,Y 433.255,Z 680.764,A -85,B 0,C 180,E1 21266.745,E2 21266.745} C_VEL
LIN {X 0,Y 433.259,Z 680.761,A -85,B 0,C 180,E1 21262.955,E2 21262.955} C_VEL
LIN {X 0,Y 433.251,Z 680.761,A -85,B 0,C 180,E1 21259.13,E2 21259.13} C_VEL
LIN {X 0,Y 433.248,Z 680.754,A -85,B 0,C 180,E1 21255.254,E2 21255.254} C_VEL
LIN {X 0,Y 433.256,Z 680.749,A -85,B 0,C 180,E1 21251.448,E2 21251.448} C_VEL
LIN {X 0,Y 433.262,Z 680.751,A -85,B 0,C 180,E1 21247.559,E2 21247.559} C_VEL
LIN {X 0,Y 433.258,Z 680.765,A -85,B 0,C 180,E1 21243.705,E2 21243.705} C_VEL
LIN {X 0,Y 433.247,Z 680.766,A -85,B 0,C 180,E1 21239.868,E2 21239.868} C_VEL
LIN {X 0,Y 433.249,Z 680.761,A -85,B 0,C 180,E1 21236.03,E2 21236.03} C_VEL
LIN {X 0,Y 433.245,Z 680.751,A -85,B 0,C 180,E1 21232.308,E2 21232.308} C_VEL
LIN {X 0,Y 433.254,Z 680.745,A -85,B 0,C 180,E1 21228.553,E2 21228.553} C_VEL
LIN {X 0,Y 433.25,Z 680.76,A -85,B 0,C 180,E1 21224.717,E2 21224.717} C_VEL
LIN {X 0,Y 433.246,Z 680.73,A -85,B 0,C 180,E1 21220.87,E2 21220.87} C_VEL
LIN {X 0,Y 433.252,Z 680.758,A -85,B 0,C 180,E1 21217.041,E2 21217.041} C_VEL
LIN {X 0,Y 433.249,Z 680.766,A -85,B 0,C 180,E1 21213.255,E2 21213.255} C_VEL
LIN {X 0,Y 433.255,Z 680.745,A -85,B 0,C 180,E1 21209.404,E2 21209.404} C_VEL
LIN {X 0,Y 433.244,Z 680.743,A -85,B 0,C 180,E1 21205.569,E2 21205.569} C_VEL
LIN {X 0,Y 433.29,Z 681.057,A -85,B 0,C 180,E1 21204.234,E2 21204.234} C_VEL
LIN {X 0,Y 434.702,Z 684.453,A -85,B 0,C 180,E1 21203.6,E2 21203.6} C_VEL
LIN {X 0,Y 435.849,Z 686.451,A -85,B 0,C 180,E1 21203.22,E2 21203.22} C_VEL
LIN {X 0,Y 442.221,Z 698.969,A -85,B 0,C 180,E1 21201.056,E2 21201.056} C_VEL
LIN {X 0,Y 450.093,Z 715.622,A -85,B 0,C 180,E1 21198.47,E2 21198.47} C_VEL
LIN {X 0,Y 458.098,Z 734.429,A -85,B 0,C 180,E1 21195.873,E2 21195.873} C_VEL
LIN {X 0,Y 459.794,Z 739.206,A -85,B 0,C 180,E1 21195.277,E2 21195.277} C_VEL
LIN {X 0,Y 459.734,Z 742.919,A -85,B 0,C 180,E1 21195.041,E2 21195.041} C_VEL
LIN {X 0,Y 466.267,Z 791.857,A -85,B 0,C 180,E1 21193.273,E2 21193.273} C_VEL
LIN {X 0,Y 460.417,Z 1020.715,A -85,B 0,C 180,E1 21189.341,E2 21189.341} C_VEL
LIN {X 0,Y 459.295,Z 1056.768,A -85,B 0,C 180,E1 21188.685,E2 21188.685} C_VEL
LIN {X 0,Y 457.696,Z 1078.804,A -85,B 0,C 180,E1 21188.096,E2 21188.096} C_VEL
LIN {X 0,Y 455.72,Z 1100.058,A -85,B 0,C 180,E1 21187.306,E2 21187.306} C_VEL
LIN {X 0,Y 453.438,Z 1121.644,A -85,B 0,C 180,E1 21186.271,E2 21186.271} C_VEL
LIN {X 0,Y 450.96,Z 1142.086,A -85,B 0,C 180,E1 21185.046,E2 21185.046} C_VEL
LIN {X 0,Y 448.317,Z 1162.235,A -85,B 0,C 180,E1 21183.579,E2 21183.579} C_VEL
LIN {X 0,Y 445.706,Z 1181.644,A -85,B 0,C 180,E1 21181.903,E2 21181.903} C_VEL
LIN {X 0,Y 443.103,Z 1200.564,A -85,B 0,C 180,E1 21179.979,E2 21179.979} C_VEL
LIN {X 0,Y 440.646,Z 1218.206,A -85,B 0,C 180,E1 21177.867,E2 21177.867} C_VEL
LIN {X 0,Y 438.438,Z 1234.976,A -85,B 0,C 180,E1 21175.531,E2 21175.531} C_VEL
LIN {X 0,Y 436.656,Z 1249.501,A -85,B 0,C 180,E1 21173.193,E2 21173.193} C_VEL
LIN {X 0,Y 435.092,Z 1263.287,A -85,B 0,C 180,E1 21170.585,E2 21170.585} C_VEL
LIN {X 0,Y 433.872,Z 1275.452,A -85,B 0,C 180,E1 21167.87,E2 21167.87} C_VEL
LIN {X 0,Y 433.005,Z 1285.791,A -85,B 0,C 180,E1 21165.125,E2 21165.125} C_VEL
LIN {X 0,Y 432.483,Z 1293.349,A -85,B 0,C 180,E1 21162.679,E2 21162.679} C_VEL
LIN {X 0,Y 432.162,Z 1299.384,A -85,B 0,C 180,E1 21160.127,E2 21160.127} C_VEL
LIN {X 0,Y 431.984,Z 1304.019,A -85,B 0,C 180,E1 21157.447,E2 21157.447} C_VEL
LIN {X 0,Y 431.918,Z 1307.444,A -85,B 0,C 180,E1 21154.514,E2 21154.514} C_VEL
LIN {X 0,Y 431.896,Z 1309.209,A -85,B 0,C 180,E1 21151.725,E2 21151.725} C_VEL
LIN {X 0,Y 431.904,Z 1309.347,A -85,B 0,C 180,E1 21149.072,E2 21149.072} C_VEL
LIN {X 0,Y 431.904,Z 1308.123,A -85,B 0,C 180,E1 21146.284,E2 21146.284} C_VEL
LIN {X 0,Y 431.946,Z 1305.455,A -85,B 0,C 180,E1 21143.621,E2 21143.621} C_VEL
LIN {X 0,Y 432.094,Z 1300.907,A -85,B 0,C 180,E1 21140.679,E2 21140.679} C_VEL
LIN {X 0,Y 432.344,Z 1295.795,A -85,B 0,C 180,E1 21138.258,E2 21138.258} C_VEL
LIN {X 0,Y 432.794,Z 1288.458,A -85,B 0,C 180,E1 21135.689,E2 21135.689} C_VEL
LIN {X 0,Y 433.568,Z 1278.886,A -85,B 0,C 180,E1 21132.97,E2 21132.97} C_VEL
LIN {X 0,Y 434.616,Z 1267.814,A -85,B 0,C 180,E1 21130.375,E2 21130.375} C_VEL
LIN {X 0,Y 436.107,Z 1254.045,A -85,B 0,C 180,E1 21127.631,E2 21127.631} C_VEL
LIN {X 0,Y 437.875,Z 1239.51,A -85,B 0,C 180,E1 21125.157,E2 21125.157} C_VEL
LIN {X 0,Y 439.968,Z 1223.451,A -85,B 0,C 180,E1 21122.821,E2 21122.821} C_VEL
LIN {X 0,Y 442.258,Z 1206.451,A -85,B 0,C 180,E1 21120.696,E2 21120.696} C_VEL
LIN {X 0,Y 444.812,Z 1188.093,A -85,B 0,C 180,E1 21118.719,E2 21118.719} C_VEL
LIN {X 0,Y 447.543,Z 1168.307,A -85,B 0,C 180,E1 21116.907,E2 21116.907} C_VEL
LIN {X 0,Y 450.152,Z 1148.427,A -85,B 0,C 180,E1 21115.389,E2 21115.389} C_VEL
LIN {X 0,Y 452.78,Z 1127,A -85,B 0,C 180,E1 21114.029,E2 21114.029} C_VEL
LIN {X 0,Y 455.154,Z 1106.128,A -85,B 0,C 180,E1 21112.955,E2 21112.955} C_VEL
LIN {X 0,Y 457.203,Z 1084.539,A -85,B 0,C 180,E1 21112.096,E2 21112.096} C_VEL
LIN {X 0,Y 458.951,Z 1061.975,A -85,B 0,C 180,E1 21111.44,E2 21111.44} C_VEL
LIN {X 0,Y 459.998,Z 1037.793,A -85,B 0,C 180,E1 21110.951,E2 21110.951} C_VEL
LIN {X 0,Y 465.59,Z 816.414,A -85,B 0,C 180,E1 21107.152,E2 21107.152} C_VEL
LIN {X 0,Y 466.129,Z 789.694,A -85,B 0,C 180,E1 21106.67,E2 21106.67} C_VEL
LIN {X 0,Y 459.615,Z 741.498,A -85,B 0,C 180,E1 21104.895,E2 21104.895} C_VEL
LIN {X 0,Y 459.656,Z 738.329,A -85,B 0,C 180,E1 21104.636,E2 21104.636} C_VEL
LIN {X 0,Y 451.449,Z 718.685,A -85,B 0,C 180,E1 21101.979,E2 21101.979} C_VEL
LIN {X 0,Y 443.741,Z 702.01,A -85,B 0,C 180,E1 21099.451,E2 21099.451} C_VEL
LIN {X 0,Y 436.894,Z 688.637,A -85,B 0,C 180,E1 21097.169,E2 21097.169} C_VEL
LIN {X 0,Y 435.095,Z 684.975,A -85,B 0,C 180,E1 21096.526,E2 21096.526} C_VEL
LIN {X 0,Y 433.335,Z 681.298,A -85,B 0,C 180,E1 21095.843,E2 21095.843} C_VEL
LIN {X 0,Y 433.246,Z 680.767,A -85,B 0,C 180,E1 21095.399,E2 21095.399} C_VEL
LIN {X 0,Y 433.252,Z 680.769,A -85,B 0,C 180,E1 21091.592,E2 21091.592} C_VEL
LIN {X 0,Y 433.251,Z 680.761,A -85,B 0,C 180,E1 21087.786,E2 21087.786} C_VEL
LIN {X 0,Y 433.247,Z 680.739,A -85,B 0,C 180,E1 21083.954,E2 21083.954} C_VEL
LIN {X 0,Y 433.248,Z 680.74,A -85,B 0,C 180,E1 21080.253,E2 21080.253} C_VEL
LIN {X 0,Y 433.249,Z 680.767,A -85,B 0,C 180,E1 21076.353,E2 21076.353} C_VEL
LIN {X 0,Y 433.249,Z 680.73,A -85,B 0,C 180,E1 21072.532,E2 21072.532} C_VEL
LIN {X 0,Y 433.245,Z 680.76,A -85,B 0,C 180,E1 21068.761,E2 21068.761} C_VEL
LIN {X 0,Y 433.258,Z 680.768,A -85,B 0,C 180,E1 21065.031,E2 21065.031} C_VEL
LIN {X 0,Y 433.249,Z 680.762,A -85,B 0,C 180,E1 21061.19,E2 21061.19} C_VEL
LIN {X 0,Y 433.251,Z 680.75,A -85,B 0,C 180,E1 21057.354,E2 21057.354} C_VEL
LIN {X 0,Y 433.245,Z 680.747,A -85,B 0,C 180,E1 21053.507,E2 21053.507} C_VEL
LIN {X 0,Y 433.258,Z 680.756,A -85,B 0,C 180,E1 21049.764,E2 21049.764} C_VEL
LIN {X 0,Y 433.262,Z 680.766,A -85,B 0,C 180,E1 21045.977,E2 21045.977} C_VEL
LIN {X 0,Y 433.259,Z 680.765,A -85,B 0,C 180,E1 21042.125,E2 21042.125} C_VEL
LIN {X 0,Y 433.248,Z 680.761,A -85,B 0,C 180,E1 21038.33,E2 21038.33} C_VEL
LIN {X 0,Y 433.253,Z 680.76,A -85,B 0,C 180,E1 21034.465,E2 21034.465} C_VEL
LIN {X 0,Y 433.25,Z 680.706,A -85,B 0,C 180,E1 21030.708,E2 21030.708} C_VEL
LIN {X 0,Y 433.256,Z 680.763,A -85,B 0,C 180,E1 21026.842,E2 21026.842} C_VEL
LIN {X 0,Y 433.247,Z 680.709,A -85,B 0,C 180,E1 21022.962,E2 21022.962} C_VEL
LIN {X 0,Y 433.247,Z 680.743,A -85,B 0,C 180,E1 21019.195,E2 21019.195} C_VEL
LIN {X 0,Y 433.285,Z 680.979,A -85,B 0,C 180,E1 21017.637,E2 21017.637} C_VEL
LIN {X 0,Y 433.687,Z 682.51,A -85,B 0,C 180,E1 21017.372,E2 21017.372} C_VEL
LIN {X 0,Y 435.714,Z 685.57,A -85,B 0,C 180,E1 21016.991,E2 21016.991} C_VEL
LIN {X 0,Y 437.243,Z 687.136,A -85,B 0,C 180,E1 21016.729,E2 21016.729} C_VEL
LIN {X 0,Y 439.918,Z 691.079,A -85,B 0,C 180,E1 21016.25,E2 21016.25} C_VEL
LIN {X 0,Y 441.579,Z 693.348,A -85,B 0,C 180,E1 21015.962,E2 21015.962} C_VEL
LIN {X 0,Y 451.658,Z 707.349,A -85,B 0,C 180,E1 21014.285,E2 21014.285} C_VEL
LIN {X 0,Y 465.271,Z 727.867,A -85,B 0,C 180,E1 21012.172,E2 21012.172} C_VEL
LIN {X 0,Y 466.204,Z 729.844,A -85,B 0,C 180,E1 21012.023,E2 21012.023} C_VEL
LIN {X 0,Y 460.766,Z 926.126,A -85,B 0,C 180,E1 21008.596,E2 21008.596} C_VEL
LIN {X 0,Y 459.65,Z 947.661,A -85,B 0,C 180,E1 21008,E2 21008} C_VEL
LIN {X 0,Y 458.319,Z 966.422,A -85,B 0,C 180,E1 21007.299,E2 21007.299} C_VEL
LIN {X 0,Y 456.886,Z 973.809,A -85,B 0,C 180,E1 21007.047,E2 21007.047} C_VEL
LIN {X 0,Y 450.315,Z 992.626,A -85,B 0,C 180,E1 21006.57,E2 21006.57} C_VEL
LIN {X 0,Y 448.732,Z 999.508,A -85,B 0,C 180,E1 21006.23,E2 21006.23} C_VEL
LIN {X 0,Y 446.118,Z 1019.268,A -85,B 0,C 180,E1 21004.855,E2 21004.855} C_VEL
LIN {X 0,Y 443.475,Z 1036.975,A -85,B 0,C 180,E1 21003.374,E2 21003.374} C_VEL
LIN {X 0,Y 440.518,Z 1054.442,A -85,B 0,C 180,E1 21001.621,E2 21001.621} C_VEL
LIN {X 0,Y 437.57,Z 1070.978,A -85,B 0,C 180,E1 20999.649,E2 20999.649} C_VEL
LIN {X 0,Y 434.768,Z 1086.09,A -85,B 0,C 180,E1 20997.531,E2 20997.531} C_VEL
LIN {X 0,Y 432.142,Z 1100.147,A -85,B 0,C 180,E1 20995.196,E2 20995.196} C_VEL
LIN {X 0,Y 429.825,Z 1112.712,A -85,B 0,C 180,E1 20992.714,E2 20992.714} C_VEL
LIN {X 0,Y 427.802,Z 1124.45,A -85,B 0,C 180,E1 20989.951,E2 20989.951} C_VEL
LIN {X 0,Y 426.302,Z 1134.189,A -85,B 0,C 180,E1 20987.188,E2 20987.188} C_VEL
LIN {X 0,Y 425.238,Z 1142.43,A -85,B 0,C 180,E1 20984.293,E2 20984.293} C_VEL
LIN {X 0,Y 424.544,Z 1148.913,A -85,B 0,C 180,E1 20981.41,E2 20981.41} C_VEL
LIN {X 0,Y 424.174,Z 1154.045,A -85,B 0,C 180,E1 20978.403,E2 20978.403} C_VEL
LIN {X 0,Y 423.998,Z 1157.442,A -85,B 0,C 180,E1 20975.548,E2 20975.548} C_VEL
LIN {X 0,Y 423.927,Z 1159.442,A -85,B 0,C 180,E1 20972.568,E2 20972.568} C_VEL
LIN {X 0,Y 423.921,Z 1160.024,A -85,B 0,C 180,E1 20969.595,E2 20969.595} C_VEL
LIN {X 0,Y 423.942,Z 1159.184,A -85,B 0,C 180,E1 20966.755,E2 20966.755} C_VEL
LIN {X 0,Y 424.019,Z 1156.823,A -85,B 0,C 180,E1 20963.773,E2 20963.773} C_VEL
LIN {X 0,Y 424.256,Z 1152.967,A -85,B 0,C 180,E1 20960.778,E2 20960.778} C_VEL
LIN {X 0,Y 424.648,Z 1147.733,A -85,B 0,C 180,E1 20957.904,E2 20957.904} C_VEL
LIN {X 0,Y 425.417,Z 1140.821,A -85,B 0,C 180,E1 20955.011,E2 20955.011} C_VEL
LIN {X 0,Y 426.599,Z 1132.131,A -85,B 0,C 180,E1 20952.098,E2 20952.098} C_VEL
LIN {X 0,Y 428.207,Z 1122.144,A -85,B 0,C 180,E1 20949.355,E2 20949.355} C_VEL
LIN {X 0,Y 430.22,Z 1110.526,A -85,B 0,C 180,E1 20946.729,E2 20946.729} C_VEL
LIN {X 0,Y 432.617,Z 1097.484,A -85,B 0,C 180,E1 20944.247,E2 20944.247} C_VEL
LIN {X 0,Y 435.267,Z 1083.458,A -85,B 0,C 180,E1 20941.982,E2 20941.982} C_VEL
LIN {X 0,Y 438.055,Z 1068.412,A -85,B 0,C 180,E1 20939.927,E2 20939.927} C_VEL
LIN {X 0,Y 440.818,Z 1052.657,A -85,B 0,C 180,E1 20938.098,E2 20938.098} C_VEL
LIN {X 0,Y 443.692,Z 1035.6,A -85,B 0,C 180,E1 20936.412,E2 20936.412} C_VEL
LIN {X 0,Y 446.35,Z 1017.677,A -85,B 0,C 180,E1 20934.931,E2 20934.931} C_VEL
LIN {X 0,Y 448.911,Z 998.063,A -85,B 0,C 180,E1 20933.59,E2 20933.59} C_VEL
LIN {X 0,Y 451.125,Z 978.261,A -85,B 0,C 180,E1 20932.492,E2 20932.492} C_VEL
LIN {X 0,Y 452.814,Z 958.705,A -85,B 0,C 180,E1 20931.641,E2 20931.641} C_VEL
LIN {X 0,Y 454.183,Z 936.593,A -85,B 0,C 180,E1 20930.919,E2 20930.919} C_VEL
LIN {X 0,Y 455.034,Z 914.279,A -85,B 0,C 180,E1 20930.425,E2 20930.425} C_VEL
LIN {X 0,Y 460.261,Z 732.777,A -85,B 0,C 180,E1 20927.245,E2 20927.245} C_VEL
LIN {X 0,Y 446.652,Z 712.101,A -85,B 0,C 180,E1 20925.068,E2 20925.068} C_VEL
LIN {X 0,Y 435.875,Z 697.185,A -85,B 0,C 180,E1 20923.215,E2 20923.215} C_VEL
LIN {X 0,Y 432.321,Z 692.337,A -85,B 0,C 180,E1 20922.57,E2 20922.57} C_VEL
LIN {X 0,Y 429.566,Z 688.478,A -85,B 0,C 180,E1 20922.054,E2 20922.054} C_VEL
LIN {X 0,Y 428.525,Z 687.185,A -85,B 0,C 180,E1 20921.86,E2 20921.86} C_VEL
LIN {X 0,Y 426.181,Z 684.457,A -85,B 0,C 180,E1 20921.422,E2 20921.422} C_VEL
LIN {X 0,Y 425.416,Z 682.341,A -85,B 0,C 180,E1 20921.154,E2 20921.154} C_VEL
LIN {X 0,Y 425.313,Z 681.763,A -85,B 0,C 180,E1 20920.803,E2 20920.803} C_VEL
LIN {X 0,Y 425.305,Z 681.695,A -85,B 0,C 180,E1 20916.938,E2 20916.938} C_VEL
LIN {X 0,Y 425.317,Z 681.75,A -85,B 0,C 180,E1 20913.052,E2 20913.052} C_VEL
LIN {X 0,Y 425.31,Z 681.692,A -85,B 0,C 180,E1 20909.274,E2 20909.274} C_VEL
LIN {X 0,Y 425.315,Z 681.748,A -85,B 0,C 180,E1 20905.481,E2 20905.481} C_VEL
LIN {X 0,Y 425.309,Z 681.75,A -85,B 0,C 180,E1 20901.66,E2 20901.66} C_VEL
LIN {X 0,Y 425.319,Z 681.753,A -85,B 0,C 180,E1 20897.795,E2 20897.795} C_VEL
LIN {X 0,Y 425.321,Z 681.756,A -85,B 0,C 180,E1 20893.874,E2 20893.874} C_VEL
LIN {X 0,Y 425.322,Z 681.747,A -85,B 0,C 180,E1 20889.948,E2 20889.948} C_VEL
LIN {X 0,Y 425.314,Z 681.737,A -85,B 0,C 180,E1 20886.073,E2 20886.073} C_VEL
LIN {X 0,Y 425.306,Z 681.736,A -85,B 0,C 180,E1 20882.291,E2 20882.291} C_VEL
LIN {X 0,Y 425.315,Z 681.747,A -85,B 0,C 180,E1 20878.518,E2 20878.518} C_VEL
LIN {X 0,Y 425.313,Z 681.756,A -85,B 0,C 180,E1 20874.604,E2 20874.604} C_VEL
LIN {X 0,Y 425.319,Z 681.752,A -85,B 0,C 180,E1 20870.802,E2 20870.802} C_VEL
LIN {X 0,Y 425.304,Z 681.715,A -85,B 0,C 180,E1 20866.957,E2 20866.957} C_VEL
LIN {X 0,Y 425.312,Z 681.753,A -85,B 0,C 180,E1 20863.052,E2 20863.052} C_VEL
LIN {X 0,Y 425.312,Z 681.739,A -85,B 0,C 180,E1 20859.208,E2 20859.208} C_VEL
LIN {X 0,Y 425.307,Z 681.723,A -85,B 0,C 180,E1 20855.411,E2 20855.411} C_VEL
LIN {X 0,Y 425.318,Z 681.732,A -85,B 0,C 180,E1 20851.496,E2 20851.496} C_VEL
LIN {X 0,Y 425.309,Z 681.75,A -85,B 0,C 180,E1 20847.748,E2 20847.748} C_VEL
LIN {X 0,Y 425.346,Z 682,A -85,B 0,C 180,E1 20845.387,E2 20845.387} C_VEL
LIN {X 0,Y 426.929,Z 685.674,A -85,B 0,C 180,E1 20844.657,E2 20844.657} C_VEL
LIN {X 0,Y 428.024,Z 687.675,A -85,B 0,C 180,E1 20844.268,E2 20844.268} C_VEL
LIN {X 0,Y 434.649,Z 700.521,A -85,B 0,C 180,E1 20841.939,E2 20841.939} C_VEL
LIN {X 0,Y 442.607,Z 717.157,A -85,B 0,C 180,E1 20839.243,E2 20839.243} C_VEL
LIN {X 0,Y 450.479,Z 735.487,A -85,B 0,C 180,E1 20836.611,E2 20836.611} C_VEL
LIN {X 0,Y 452.827,Z 740.961,A -85,B 0,C 180,E1 20835.931,E2 20835.931} C_VEL
LIN {X 0,Y 453.771,Z 743.258,A -85,B 0,C 180,E1 20835.76,E2 20835.76} C_VEL
LIN {X 0,Y 460.3,Z 793.281,A -85,B 0,C 180,E1 20833.917,E2 20833.917} C_VEL
LIN {X 0,Y 454.108,Z 1021.825,A -85,B 0,C 180,E1 20829.946,E2 20829.946} C_VEL
LIN {X 0,Y 452.962,Z 1055.84,A -85,B 0,C 180,E1 20829.314,E2 20829.314} C_VEL
LIN {X 0,Y 451.306,Z 1077.629,A -85,B 0,C 180,E1 20828.725,E2 20828.725} C_VEL
LIN {X 0,Y 449.14,Z 1099.372,A -85,B 0,C 180,E1 20827.908,E2 20827.908} C_VEL
LIN {X 0,Y 446.709,Z 1120.887,A -85,B 0,C 180,E1 20826.858,E2 20826.858} C_VEL
LIN {X 0,Y 444.146,Z 1140.921,A -85,B 0,C 180,E1 20825.642,E2 20825.642} C_VEL
LIN {X 0,Y 441.358,Z 1160.757,A -85,B 0,C 180,E1 20824.181,E2 20824.181} C_VEL
LIN {X 0,Y 438.606,Z 1180.064,A -85,B 0,C 180,E1 20822.493,E2 20822.493} C_VEL
LIN {X 0,Y 435.89,Z 1198.363,A -85,B 0,C 180,E1 20820.612,E2 20820.612} C_VEL
LIN {X 0,Y 433.355,Z 1215.638,A -85,B 0,C 180,E1 20818.528,E2 20818.528} C_VEL
LIN {X 0,Y 430.973,Z 1232.582,A -85,B 0,C 180,E1 20816.154,E2 20816.154} C_VEL
LIN {X 0,Y 429.048,Z 1247.225,A -85,B 0,C 180,E1 20813.775,E2 20813.775} C_VEL
LIN {X 0,Y 427.434,Z 1260.436,A -85,B 0,C 180,E1 20811.258,E2 20811.258} C_VEL
LIN {X 0,Y 426.092,Z 1272.955,A -85,B 0,C 180,E1 20808.468,E2 20808.468} C_VEL
LIN {X 0,Y 425.156,Z 1283.446,A -85,B 0,C 180,E1 20805.691,E2 20805.691} C_VEL
LIN {X 0,Y 424.555,Z 1291.914,A -85,B 0,C 180,E1 20802.928,E2 20802.928} C_VEL
LIN {X 0,Y 424.173,Z 1298.973,A -85,B 0,C 180,E1 20800.045,E2 20800.045} C_VEL
LIN {X 0,Y 423.988,Z 1303.793,A -85,B 0,C 180,E1 20797.452,E2 20797.452} C_VEL
LIN {X 0,Y 423.919,Z 1307.201,A -85,B 0,C 180,E1 20794.735,E2 20794.735} C_VEL
LIN {X 0,Y 423.906,Z 1308.977,A -85,B 0,C 180,E1 20792.163,E2 20792.163} C_VEL
LIN {X 0,Y 423.898,Z 1309.367,A -85,B 0,C 180,E1 20789.324,E2 20789.324} C_VEL
LIN {X 0,Y 423.909,Z 1308.334,A -85,B 0,C 180,E1 20786.62,E2 20786.62} C_VEL
LIN {X 0,Y 423.935,Z 1305.691,A -85,B 0,C 180,E1 20783.908,E2 20783.908} C_VEL
LIN {X 0,Y 424.054,Z 1301.718,A -85,B 0,C 180,E1 20781.321,E2 20781.321} C_VEL
LIN {X 0,Y 424.33,Z 1295.839,A -85,B 0,C 180,E1 20778.584,E2 20778.584} C_VEL
LIN {X 0,Y 424.786,Z 1288.35,A -85,B 0,C 180,E1 20775.831,E2 20775.831} C_VEL
LIN {X 0,Y 425.546,Z 1278.944,A -85,B 0,C 180,E1 20773.062,E2 20773.062} C_VEL
LIN {X 0,Y 426.646,Z 1267.593,A -85,B 0,C 180,E1 20770.278,E2 20770.278} C_VEL
LIN {X 0,Y 428.088,Z 1254.835,A -85,B 0,C 180,E1 20767.623,E2 20767.623} C_VEL
LIN {X 0,Y 429.894,Z 1240.582,A -85,B 0,C 180,E1 20765.103,E2 20765.103} C_VEL
LIN {X 0,Y 432.065,Z 1224.734,A -85,B 0,C 180,E1 20762.701,E2 20762.701} C_VEL
LIN {X 0,Y 434.579,Z 1207.25,A -85,B 0,C 180,E1 20760.421,E2 20760.421} C_VEL
LIN {X 0,Y 437.302,Z 1188.968,A -85,B 0,C 180,E1 20758.379,E2 20758.379} C_VEL
LIN {X 0,Y 440.094,Z 1169.751,A -85,B 0,C 180,E1 20756.57,E2 20756.57} C_VEL
LIN {X 0,Y 442.869,Z 1150.189,A -85,B 0,C 180,E1 20755.01,E2 20755.01} C_VEL
LIN {X 0,Y 445.546,Z 1130.194,A -85,B 0,C 180,E1 20753.67,E2 20753.67} C_VEL
LIN {X 0,Y 448.063,Z 1109.386,A -85,B 0,C 180,E1 20752.55,E2 20752.55} C_VEL
LIN {X 0,Y 450.407,Z 1087.165,A -85,B 0,C 180,E1 20751.607,E2 20751.607} C_VEL
LIN {X 0,Y 452.295,Z 1065.655,A -85,B 0,C 180,E1 20750.923,E2 20750.923} C_VEL
LIN {X 0,Y 453.525,Z 1042.976,A -85,B 0,C 180,E1 20750.425,E2 20750.425} C_VEL
LIN {X 0,Y 459.469,Z 821.863,A -85,B 0,C 180,E1 20746.584,E2 20746.584} C_VEL
LIN {X 0,Y 460.162,Z 791.143,A -85,B 0,C 180,E1 20746.026,E2 20746.026} C_VEL
LIN {X 0,Y 453.56,Z 742.373,A -85,B 0,C 180,E1 20744.199,E2 20744.199} C_VEL
LIN {X 0,Y 451.758,Z 738.694,A -85,B 0,C 180,E1 20743.821,E2 20743.821} C_VEL
LIN {X 0,Y 443.735,Z 719.678,A -85,B 0,C 180,E1 20741.144,E2 20741.144} C_VEL
LIN {X 0,Y 436.149,Z 703.441,A -85,B 0,C 180,E1 20738.576,E2 20738.576} C_VEL
LIN {X 0,Y 429.452,Z 690.367,A -85,B 0,C 180,E1 20736.254,E2 20736.254} C_VEL
LIN {X 0,Y 426.896,Z 685.629,A -85,B 0,C 180,E1 20735.346,E2 20735.346} C_VEL
LIN {X 0,Y 425.343,Z 681.98,A -85,B 0,C 180,E1 20734.613,E2 20734.613} C_VEL
LIN {X 0,Y 425.314,Z 681.738,A -85,B 0,C 180,E1 20730.903,E2 20730.903} C_VEL
LIN {X 0,Y 425.31,Z 681.759,A -85,B 0,C 180,E1 20726.982,E2 20726.982} C_VEL
LIN {X 0,Y 425.317,Z 681.741,A -85,B 0,C 180,E1 20723.116,E2 20723.116} C_VEL
LIN {X 0,Y 425.304,Z 681.718,A -85,B 0,C 180,E1 20719.358,E2 20719.358} C_VEL
LIN {X 0,Y 425.315,Z 681.75,A -85,B 0,C 180,E1 20715.458,E2 20715.458} C_VEL
LIN {X 0,Y 425.307,Z 681.73,A -85,B 0,C 180,E1 20711.664,E2 20711.664} C_VEL
LIN {X 0,Y 425.31,Z 681.739,A -85,B 0,C 180,E1 20707.837,E2 20707.837} C_VEL
LIN {X 0,Y 425.309,Z 681.75,A -85,B 0,C 180,E1 20704.044,E2 20704.044} C_VEL
LIN {X 0,Y 425.309,Z 681.755,A -85,B 0,C 180,E1 20700.134,E2 20700.134} C_VEL
LIN {X 0,Y 425.318,Z 681.755,A -85,B 0,C 180,E1 20696.226,E2 20696.226} C_VEL
LIN {X 0,Y 425.326,Z 681.74,A -85,B 0,C 180,E1 20692.299,E2 20692.299} C_VEL
LIN {X 0,Y 425.315,Z 681.737,A -85,B 0,C 180,E1 20688.473,E2 20688.473} C_VEL
LIN {X 0,Y 425.313,Z 681.74,A -85,B 0,C 180,E1 20684.594,E2 20684.594} C_VEL
LIN {X 0,Y 425.311,Z 681.748,A -85,B 0,C 180,E1 20680.784,E2 20680.784} C_VEL
LIN {X 0,Y 425.322,Z 681.749,A -85,B 0,C 180,E1 20676.884,E2 20676.884} C_VEL
LIN {X 0,Y 425.318,Z 681.75,A -85,B 0,C 180,E1 20672.992,E2 20672.992} C_VEL
LIN {X 0,Y 425.317,Z 681.689,A -85,B 0,C 180,E1 20669.097,E2 20669.097} C_VEL
LIN {X 0,Y 425.308,Z 681.737,A -85,B 0,C 180,E1 20665.325,E2 20665.325} C_VEL
LIN {X 0,Y 425.307,Z 681.715,A -85,B 0,C 180,E1 20661.465,E2 20661.465} C_VEL
LIN {X 0,Y 425.335,Z 681.932,A -85,B 0,C 180,E1 20658.875,E2 20658.875} C_VEL
LIN {X 0,Y 425.7,Z 683.363,A -85,B 0,C 180,E1 20658.588,E2 20658.588} C_VEL
LIN {X 0,Y 427.582,Z 686.372,A -85,B 0,C 180,E1 20658.207,E2 20658.207} C_VEL
LIN {X 0,Y 429.381,Z 688.097,A -85,B 0,C 180,E1 20657.883,E2 20657.883} C_VEL
LIN {X 0,Y 431.954,Z 691.975,A -85,B 0,C 180,E1 20657.394,E2 20657.394} C_VEL
LIN {X 0,Y 433.623,Z 694.045,A -85,B 0,C 180,E1 20657.094,E2 20657.094} C_VEL
LIN {X 0,Y 444.855,Z 709.664,A -85,B 0,C 180,E1 20655.132,E2 20655.132} C_VEL
LIN {X 0,Y 456.212,Z 726.502,A -85,B 0,C 180,E1 20653.289,E2 20653.289} C_VEL
LIN {X 0,Y 460.297,Z 733.128,A -85,B 0,C 180,E1 20652.65,E2 20652.65} C_VEL
LIN {X 0,Y 454.615,Z 927.444,A -85,B 0,C 180,E1 20649.22,E2 20649.22} C_VEL
LIN {X 0,Y 453.461,Z 948.978,A -85,B 0,C 180,E1 20648.617,E2 20648.617} C_VEL
LIN {X 0,Y 451.861,Z 970.069,A -85,B 0,C 180,E1 20647.8,E2 20647.8} C_VEL
LIN {X 0,Y 450.004,Z 988.801,A -85,B 0,C 180,E1 20646.862,E2 20646.862} C_VEL
LIN {X 0,Y 448.732,Z 999.508,A -85,B 0,C 180,E1 20646.23,E2 20646.23} C_VEL
LIN {X 0,Y 447.109,Z 1006.563,A -85,B 0,C 180,E1 20645.863,E2 20645.863} C_VEL
LIN {X 0,Y 439.911,Z 1024.326,A -85,B 0,C 180,E1 20645.074,E2 20645.074} C_VEL
LIN {X 0,Y 438.08,Z 1030.915,A -85,B 0,C 180,E1 20644.604,E2 20644.604} C_VEL
